Yaskawa INFORM job: u_tourne3TRJ3.JBI

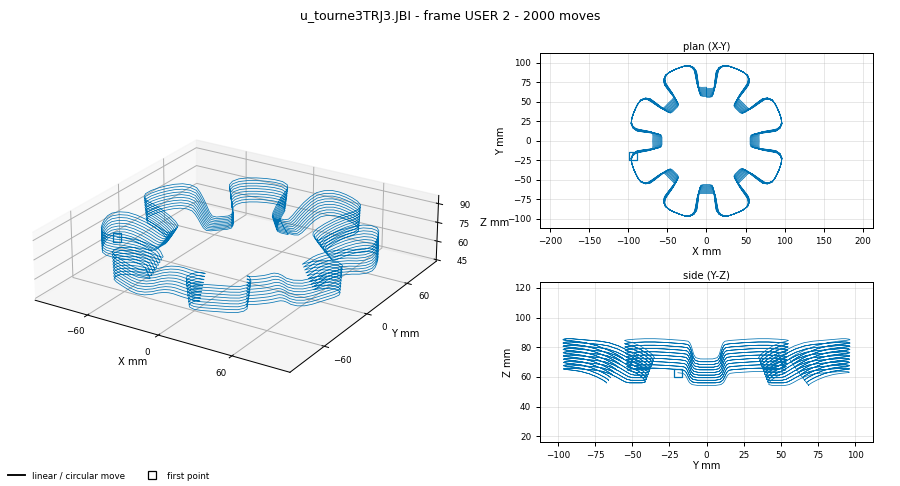
[picture p0: tool path of u_tourne3TRJ3.JBI in frame USER 2, 2000 of 2000 moves have a stored position in this frame; points joined in program order, loops and branches not executed]
/JOB
//NAME u_tourne3TRJ3
///FOLDERNAME DEMO
//POS
///NPOS 2000,0,2000,0,0,0
///USER 2
///TOOL 7
///POSTYPE USER
///RECTAN
///RCONF 1,0,0,0,0,0,0,0,0,0,0,0,0,0,0,0,0,0,0,0,0,0,0,0
C00000=-94.423,-19.246,62.877,176.5198,-3.5287,-10788.4794
C00001=-90.636,-15.942,62.469,172.2266,-2.1131,-10790.0243
C00002=-85.405,-14.621,61.698,172.0565,-0.4508,-10790.2854
C00003=-79.780,-13.569,60.151,173.8939,-0.2961,-10790.3475
C00004=-74.809,-12.586,58.158,176.9112,-0.2537,-10790.4499
C00005=-71.127,-11.507,56.252,-176.4195,0.6994,-10790.8103
C00006=-69.044,-9.699,54.888,-160.3569,24.2302,-10792.0037
C00007=-68.619,-6.200,54.350,-174.8933,38.1355,-10794.8371
C00008=-68.781,-2.945,54.326,179.7056,38.7871,-10797.5483
C00009=-68.843,0.000,54.342,180.0000,38.7770,-10800.0000
C00010=-68.781,2.945,54.326,-179.7056,38.7871,-10802.4517
C00011=-68.619,6.200,54.350,174.8933,38.1355,-10805.1629
C00012=-69.044,9.699,54.888,160.3561,24.2357,-10807.9963
C00013=-71.127,11.507,56.252,176.4195,0.6994,-10809.1897
C00014=-74.809,12.586,58.158,-176.9112,-0.2537,-10809.5501
C00015=-79.780,13.569,60.151,-173.8939,-0.2961,-10809.6525
C00016=-85.405,14.621,61.698,-172.0565,-0.4508,-10809.7146
C00017=-90.636,15.942,62.469,-172.2266,-2.1131,-10809.9757
C00018=-94.423,19.246,62.877,-176.5198,-3.5287,-10811.5206
C00019=-96.154,24.159,63.210,-179.1544,-2.3288,-10814.1038
C00020=-95.429,29.718,63.547,-179.9995,-0.1559,-10817.2974
C00021=-93.512,35.416,63.770,-179.9993,-0.0181,-10820.7433
C00022=-91.166,41.080,63.770,-179.9982,-0.0180,-10824.2566
C00023=-88.493,46.465,63.547,179.9980,-0.1564,-10827.7026
C00024=-85.074,50.908,63.210,179.1554,-2.3286,-10830.8962
C00025=-80.376,53.158,62.877,176.5237,-3.5316,-10833.4793
C00026=-75.362,52.817,62.469,172.2314,-2.1139,-10835.0245
C00027=-70.729,50.052,61.698,172.0558,-0.4490,-10835.2855
C00028=-66.007,46.818,60.151,173.8890,-0.2958,-10835.3476
C00029=-61.798,43.998,58.158,176.9122,-0.2494,-10835.4495
C00030=-58.431,42.158,56.252,-176.4248,0.6998,-10835.8105
C00031=-55.679,41.963,54.888,-160.3550,24.2338,-10837.0038
C00032=-52.905,44.137,54.350,-174.8913,38.1376,-10839.8372
C00033=-50.718,46.553,54.326,179.7087,38.7878,-10842.5482
C00034=-48.679,48.679,54.342,179.9948,38.7763,-10845.0000
C00035=-46.553,50.718,54.326,-179.7087,38.7878,-10847.4518
C00036=-44.137,52.905,54.350,174.8913,38.1376,-10850.1628
C00037=-41.963,55.680,54.888,160.3548,24.2336,-10852.9966
C00038=-42.158,58.431,56.252,176.4248,0.6998,-10854.1895
C00039=-43.998,61.798,58.158,-176.9122,-0.2494,-10854.5505
C00040=-46.818,66.007,60.151,-173.8890,-0.2958,-10854.6524
C00041=-50.052,70.729,61.698,-172.0558,-0.4490,-10854.7145
C00042=-52.817,75.362,62.469,-172.2314,-2.1139,-10854.9755
C00043=-53.158,80.376,62.877,-176.5237,-3.5316,-10856.5207
C00044=-50.908,85.074,63.210,-179.1554,-2.3286,-10859.1038
C00045=-46.465,88.493,63.547,-179.9980,-0.1564,-10862.2974
C00046=-41.080,91.166,63.770,179.9982,-0.0180,-10865.7434
C00047=-35.416,93.512,63.770,179.9993,-0.0181,-10869.2567
C00048=-29.718,95.429,63.547,179.9995,-0.1559,-10872.7026
C00049=-24.159,96.154,63.210,179.1544,-2.3288,-10875.8962
C00050=-19.246,94.423,62.877,176.5198,-3.5287,-10878.4794
C00051=-15.942,90.636,62.469,172.2266,-2.1131,-10880.0243
C00052=-14.621,85.405,61.698,172.0565,-0.4508,-10880.2854
C00053=-13.569,79.780,60.151,173.8939,-0.2961,-10880.3475
C00054=-12.586,74.809,58.158,176.9112,-0.2537,-10880.4499
C00055=-11.507,71.127,56.252,-176.4195,0.6994,-10880.8103
C00056=-9.699,69.044,54.888,-160.3561,24.2357,-10882.0037
C00057=-6.200,68.619,54.350,-174.8933,38.1355,-10884.8371
C00058=-2.945,68.781,54.326,179.7056,38.7871,-10887.5483
C00059=0.000,68.843,54.342,180.0000,38.7770,-10890.0000
C00060=0.000,67.469,56.061,180.0000,38.4594,-10890.0000
C00061=2.820,67.413,56.044,-179.6998,38.4717,-10892.3954
C00062=5.989,67.263,56.069,174.6494,37.7561,-10895.0881
C00063=9.441,67.734,56.637,160.4399,22.8847,-10897.9350
C00064=11.191,69.937,58.076,177.3917,0.4478,-10899.0911
C00065=12.227,73.809,60.085,-176.5319,-0.2393,-10899.4060
C00066=13.183,79.025,62.181,-173.7887,-0.2511,-10899.4709
C00067=14.211,84.918,63.804,-172.0889,-0.3684,-10899.5004
C00068=15.500,90.396,64.610,-172.2474,-1.9783,-10899.7298
C00069=18.832,94.373,65.037,-176.4691,-3.4890,-10901.2851
C00070=23.832,96.213,65.385,-179.1427,-2.3150,-10903.9122
C00071=29.513,95.497,65.736,-179.9981,-0.1613,-10907.1736
C00072=35.347,93.539,65.969,-179.9993,-0.0181,-10910.7008
C00073=41.148,91.136,65.969,-179.9981,-0.0180,-10914.2992
C00074=46.658,88.395,65.736,179.9983,-0.1564,-10917.8267
C00075=51.181,84.885,65.385,179.1465,-2.3148,-10921.0877
C00076=53.416,80.048,65.037,176.4667,-3.4903,-10923.7152
C00077=52.959,74.880,64.610,172.2446,-1.9818,-10925.2699
C00078=49.997,70.095,63.804,172.0881,-0.3719,-10925.4993
C00079=46.557,65.200,62.181,173.7887,-0.2530,-10925.5293
C00080=43.545,60.837,60.085,176.5334,-0.2396,-10925.5938
C00081=41.540,57.367,58.076,-177.3875,0.4483,-10925.9087
C00082=41.220,54.571,56.637,-160.4399,22.8842,-10927.0654
C00083=43.327,51.796,56.069,-174.6518,37.7544,-10929.9123
C00084=45.674,49.662,56.044,179.7031,38.4687,-10932.6047
C00085=47.708,47.708,56.061,-180.0000,38.4581,-10935.0000
C00086=49.662,45.674,56.044,-179.7031,38.4687,-10937.3953
C00087=51.797,43.327,56.069,174.6514,37.7543,-10940.0883
C00088=54.571,41.220,56.637,160.4399,22.8842,-10942.9346
C00089=57.367,41.540,58.076,177.3875,0.4483,-10944.0913
C00090=60.837,43.545,60.085,-176.5334,-0.2396,-10944.4062
C00091=65.200,46.557,62.181,-173.7887,-0.2530,-10944.4707
C00092=70.095,49.997,63.804,-172.0881,-0.3719,-10944.5007
C00093=74.880,52.959,64.610,-172.2446,-1.9818,-10944.7301
C00094=80.048,53.416,65.037,-176.4667,-3.4903,-10946.2848
C00095=84.885,51.181,65.385,-179.1465,-2.3148,-10948.9123
C00096=88.395,46.658,65.736,-179.9983,-0.1564,-10952.1733
C00097=91.136,41.148,65.969,179.9981,-0.0180,-10955.7008
C00098=93.539,35.347,65.969,179.9993,-0.0181,-10959.2992
C00099=95.497,29.513,65.736,179.9981,-0.1613,-10962.8264
C00100=96.213,23.832,65.385,179.1427,-2.3150,-10966.0878
C00101=94.373,18.832,65.037,176.4691,-3.4890,-10968.7149
C00102=90.396,15.500,64.610,172.2474,-1.9783,-10970.2702
C00103=84.918,14.211,63.804,172.0889,-0.3684,-10970.4996
C00104=79.025,13.183,62.181,173.7887,-0.2511,-10970.5291
C00105=73.809,12.227,60.085,176.5319,-0.2393,-10970.5940
C00106=69.937,11.191,58.076,-177.3917,0.4478,-10970.9089
C00107=67.734,9.441,56.637,-160.4399,22.8847,-10972.0650
C00108=67.263,5.989,56.069,-174.6494,37.7561,-10974.9119
C00109=67.413,2.820,56.044,179.6998,38.4717,-10977.6046
C00110=67.469,0.000,56.061,-180.0000,38.4594,-10980.0000
C00111=67.413,-2.820,56.044,-179.6998,38.4717,-10982.3954
C00112=67.263,-5.989,56.069,174.6494,37.7561,-10985.0881
C00113=67.734,-9.441,56.637,160.4399,22.8847,-10987.9350
C00114=69.937,-11.191,58.076,177.3917,0.4478,-10989.0911
C00115=73.809,-12.227,60.085,-176.5319,-0.2393,-10989.4060
C00116=79.025,-13.183,62.181,-173.7887,-0.2511,-10989.4709
C00117=84.918,-14.211,63.804,-172.0889,-0.3684,-10989.5004
C00118=90.396,-15.500,64.610,-172.2474,-1.9783,-10989.7298
C00119=94.373,-18.832,65.037,-176.4691,-3.4890,-10991.2851
C00120=96.213,-23.832,65.385,-179.1427,-2.3150,-10993.9122
C00121=95.497,-29.513,65.736,-179.9981,-0.1613,-10997.1736
C00122=93.539,-35.347,65.969,-179.9993,-0.0181,-11000.7008
C00123=91.136,-41.148,65.969,-179.9981,-0.0180,-11004.2992
C00124=88.395,-46.658,65.736,179.9983,-0.1564,-11007.8267
C00125=84.885,-51.181,65.385,179.1465,-2.3148,-11011.0877
C00126=80.048,-53.416,65.037,176.4667,-3.4903,-11013.7152
C00127=74.880,-52.959,64.610,172.2446,-1.9818,-11015.2699
C00128=70.095,-49.997,63.804,172.0881,-0.3719,-11015.4993
C00129=65.200,-46.557,62.181,173.7887,-0.2530,-11015.5293
C00130=60.837,-43.545,60.085,176.5334,-0.2396,-11015.5938
C00131=57.367,-41.540,58.076,-177.3875,0.4483,-11015.9087
C00132=54.571,-41.220,56.637,-160.4399,22.8842,-11017.0654
C00133=51.796,-43.327,56.069,-174.6518,37.7544,-11019.9123
C00134=49.662,-45.674,56.044,179.7031,38.4687,-11022.6047
C00135=47.708,-47.708,56.061,-180.0000,38.4581,-11025.0000
C00136=45.674,-49.662,56.044,-179.7031,38.4687,-11027.3953
C00137=43.327,-51.797,56.069,174.6514,37.7543,-11030.0883
C00138=41.220,-54.571,56.637,160.4399,22.8842,-11032.9346
C00139=41.540,-57.367,58.076,177.3875,0.4483,-11034.0913
C00140=43.545,-60.837,60.085,-176.5334,-0.2396,-11034.4062
C00141=46.557,-65.200,62.181,-173.7887,-0.2530,-11034.4707
C00142=49.997,-70.095,63.804,-172.0881,-0.3719,-11034.5007
C00143=52.959,-74.880,64.610,-172.2446,-1.9818,-11034.7301
C00144=53.416,-80.048,65.037,-176.4667,-3.4903,-11036.2848
C00145=51.181,-84.885,65.385,-179.1465,-2.3148,-11038.9123
C00146=46.658,-88.395,65.736,-179.9983,-0.1564,-11042.1733
C00147=41.148,-91.136,65.969,179.9981,-0.0180,-11045.7008
C00148=35.347,-93.539,65.969,179.9993,-0.0181,-11049.2992
C00149=29.513,-95.497,65.736,179.9981,-0.1613,-11052.8264
C00150=23.832,-96.213,65.385,179.1427,-2.3150,-11056.0878
C00151=18.832,-94.373,65.037,176.4691,-3.4890,-11058.7149
C00152=15.500,-90.396,64.610,172.2474,-1.9783,-11060.2702
C00153=14.211,-84.918,63.804,172.0889,-0.3684,-11060.4996
C00154=13.183,-79.025,62.181,173.7887,-0.2511,-11060.5291
C00155=12.227,-73.809,60.085,176.5319,-0.2393,-11060.5940
C00156=11.191,-69.937,58.076,-177.3917,0.4478,-11060.9089
C00157=9.441,-67.734,56.637,-160.4399,22.8847,-11062.0650
C00158=5.989,-67.263,56.069,-174.6494,37.7561,-11064.9119
C00159=2.820,-67.413,56.044,179.6998,38.4717,-11067.6046
C00160=0.000,-67.469,56.061,-180.0000,38.4594,-11070.0000
C00161=0.000,-67.469,56.061,-180.0000,38.4594,-11070.0000
C00162=-2.820,-67.413,56.044,-179.6998,38.4717,-11072.3954
C00163=-5.989,-67.263,56.069,174.6494,37.7561,-11075.0881
C00164=-9.441,-67.734,56.637,160.4399,22.8847,-11077.9350
C00165=-11.191,-69.937,58.076,177.3917,0.4478,-11079.0911
C00166=-12.227,-73.809,60.085,-176.5319,-0.2393,-11079.4060
C00167=-13.183,-79.025,62.181,-173.7887,-0.2511,-11079.4709
C00168=-14.211,-84.918,63.804,-172.0889,-0.3684,-11079.5004
C00169=-15.500,-90.396,64.610,-172.2474,-1.9783,-11079.7298
C00170=-18.832,-94.373,65.037,-176.4691,-3.4890,-11081.2851
C00171=-23.832,-96.213,65.385,-179.1427,-2.3150,-11083.9122
C00172=-29.513,-95.497,65.736,-179.9981,-0.1613,-11087.1736
C00173=-35.347,-93.539,65.969,-179.9993,-0.0181,-11090.7008
C00174=-41.148,-91.136,65.969,-179.9981,-0.0180,-11094.2992
C00175=-46.658,-88.395,65.736,179.9983,-0.1564,-11097.8267
C00176=-51.181,-84.885,65.385,179.1465,-2.3148,-11101.0877
C00177=-53.416,-80.048,65.037,176.4667,-3.4903,-11103.7152
C00178=-52.959,-74.880,64.610,172.2446,-1.9818,-11105.2699
C00179=-49.997,-70.095,63.804,172.0881,-0.3719,-11105.4993
C00180=-46.557,-65.200,62.181,173.7887,-0.2530,-11105.5293
C00181=-43.545,-60.837,60.085,176.5334,-0.2396,-11105.5938
C00182=-41.540,-57.367,58.076,-177.3875,0.4483,-11105.9087
C00183=-41.220,-54.571,56.637,-160.4399,22.8842,-11107.0654
C00184=-43.327,-51.796,56.069,-174.6518,37.7544,-11109.9123
C00185=-45.674,-49.662,56.044,179.7031,38.4687,-11112.6047
C00186=-47.708,-47.708,56.061,-180.0000,38.4581,-11115.0000
C00187=-49.662,-45.674,56.044,-179.7031,38.4687,-11117.3953
C00188=-51.797,-43.327,56.069,174.6514,37.7543,-11120.0883
C00189=-54.571,-41.220,56.637,160.4399,22.8842,-11122.9346
C00190=-57.367,-41.540,58.076,177.3875,0.4483,-11124.0913
C00191=-60.837,-43.545,60.085,-176.5334,-0.2396,-11124.4062
C00192=-65.200,-46.557,62.181,-173.7887,-0.2530,-11124.4707
C00193=-70.095,-49.997,63.804,-172.0881,-0.3719,-11124.5007
C00194=-74.880,-52.959,64.610,-172.2446,-1.9818,-11124.7301
C00195=-80.048,-53.416,65.037,-176.4667,-3.4903,-11126.2848
C00196=-84.885,-51.181,65.385,-179.1465,-2.3148,-11128.9123
C00197=-88.395,-46.658,65.736,-179.9983,-0.1564,-11132.1733
C00198=-91.136,-41.148,65.969,179.9981,-0.0180,-11135.7008
C00199=-93.539,-35.347,65.969,179.9993,-0.0181,-11139.2992
C00200=-95.497,-29.513,65.736,179.9981,-0.1613,-11142.8264
C00201=-96.213,-23.832,65.385,179.1427,-2.3150,-11146.0878
C00202=-94.373,-18.832,65.037,176.4691,-3.4890,-11148.7149
C00203=-90.396,-15.500,64.610,172.2474,-1.9783,-11150.2702
C00204=-84.918,-14.211,63.804,172.0889,-0.3684,-11150.4996
C00205=-79.025,-13.183,62.181,173.7887,-0.2511,-11150.5291
C00206=-73.809,-12.227,60.085,176.5319,-0.2393,-11150.5940
C00207=-69.937,-11.191,58.076,-177.3917,0.4478,-11150.9089
C00208=-67.734,-9.441,56.637,-160.4399,22.8847,-11152.0650
C00209=-67.263,-5.989,56.069,-174.6494,37.7561,-11154.9119
C00210=-67.413,-2.820,56.044,179.6998,38.4717,-11157.6046
C00211=-67.469,0.000,56.061,-180.0000,38.4594,-11160.0000
C00212=-67.413,2.820,56.044,-179.6998,38.4717,-11162.3954
C00213=-67.263,5.989,56.069,174.6494,37.7561,-11165.0881
C00214=-67.734,9.441,56.637,160.4399,22.8847,-11167.9350
C00215=-69.937,11.191,58.076,177.3917,0.4478,-11169.0911
C00216=-73.809,12.227,60.085,-176.5319,-0.2393,-11169.4060
C00217=-79.025,13.183,62.181,-173.7887,-0.2511,-11169.4709
C00218=-84.918,14.211,63.804,-172.0889,-0.3684,-11169.5004
C00219=-90.396,15.500,64.610,-172.2474,-1.9783,-11169.7298
C00220=-94.373,18.832,65.037,-176.4691,-3.4890,-11171.2851
C00221=-96.213,23.832,65.385,-179.1427,-2.3150,-11173.9122
C00222=-95.497,29.513,65.736,-179.9981,-0.1613,-11177.1736
C00223=-93.539,35.347,65.969,-179.9993,-0.0181,-11180.7008
C00224=-91.136,41.148,65.969,-179.9981,-0.0180,-11184.2992
C00225=-88.395,46.658,65.736,179.9983,-0.1564,-11187.8267
C00226=-84.885,51.181,65.385,179.1465,-2.3148,-11191.0877
C00227=-80.048,53.416,65.037,176.4667,-3.4903,-11193.7152
C00228=-74.880,52.959,64.610,172.2446,-1.9818,-11195.2699
C00229=-70.095,49.997,63.804,172.0881,-0.3719,-11195.4993
C00230=-65.200,46.557,62.181,173.7887,-0.2530,-11195.5293
C00231=-60.837,43.545,60.085,176.5334,-0.2396,-11195.5938
C00232=-57.367,41.540,58.076,-177.3875,0.4483,-11195.9087
C00233=-54.571,41.220,56.637,-160.4399,22.8842,-11197.0654
C00234=-51.796,43.327,56.069,-174.6518,37.7544,-11199.9123
C00235=-49.662,45.674,56.044,179.7031,38.4687,-11202.6047
C00236=-47.708,47.708,56.061,-180.0000,38.4581,-11205.0000
C00237=-45.674,49.662,56.044,-179.7031,38.4687,-11207.3953
C00238=-43.327,51.797,56.069,174.6514,37.7543,-11210.0883
C00239=-41.220,54.571,56.637,160.4399,22.8842,-11212.9346
C00240=-41.540,57.367,58.076,177.3875,0.4483,-11214.0913
C00241=-43.545,60.837,60.085,-176.5334,-0.2396,-11214.4062
C00242=-46.557,65.200,62.181,-173.7887,-0.2530,-11214.4707
C00243=-49.997,70.095,63.804,-172.0881,-0.3719,-11214.5007
C00244=-52.959,74.880,64.610,-172.2446,-1.9818,-11214.7301
C00245=-53.416,80.048,65.037,-176.4667,-3.4903,-11216.2848
C00246=-51.181,84.885,65.385,-179.1465,-2.3148,-11218.9123
C00247=-46.658,88.395,65.736,-179.9983,-0.1564,-11222.1733
C00248=-41.148,91.136,65.969,179.9981,-0.0180,-11225.7008
C00249=-35.347,93.539,65.969,179.9993,-0.0181,-11229.2992
C00250=-29.513,95.497,65.736,179.9981,-0.1613,-11232.8264
C00251=-23.832,96.213,65.385,179.1427,-2.3150,-11236.0878
C00252=-18.832,94.373,65.037,176.4691,-3.4890,-11238.7149
C00253=-15.500,90.396,64.610,172.2474,-1.9783,-11240.2702
C00254=-14.211,84.918,63.804,172.0889,-0.3684,-11240.4996
C00255=-13.183,79.025,62.181,173.7887,-0.2511,-11240.5291
C00256=-12.227,73.809,60.085,176.5319,-0.2393,-11240.5940
C00257=-11.191,69.937,58.076,-177.3917,0.4478,-11240.9089
C00258=-9.441,67.734,56.637,-160.4399,22.8847,-11242.0650
C00259=-5.989,67.263,56.069,-174.6494,37.7561,-11244.9119
C00260=-2.820,67.413,56.044,179.6998,38.4717,-11247.6046
C00261=0.000,67.469,56.061,180.0000,38.4594,-11250.0000
C00262=0.000,66.107,57.788,180.0000,38.0594,-11250.0000
C00263=2.695,66.055,57.771,-179.6967,38.0667,-11252.3363
C00264=5.779,65.917,57.797,174.4231,37.2903,-11255.0104
C00265=9.185,66.436,58.394,160.6412,21.4973,-11257.8714
C00266=10.880,68.762,59.909,178.2705,0.2602,-11258.9912
C00267=11.874,72.826,62.021,-176.2283,-0.2219,-11259.2604
C00268=12.805,78.288,64.219,-173.7529,-0.2122,-11259.2892
C00269=13.814,84.445,65.915,-172.1933,-0.3031,-11259.2905
C00270=15.073,90.163,66.756,-172.3373,-1.8422,-11259.4907
C00271=18.432,94.325,67.200,-176.4590,-3.4166,-11261.0568
C00272=23.517,96.271,67.561,-179.1417,-2.2803,-11263.7273
C00273=29.315,95.562,67.927,179.9999,-0.1559,-11267.0541
C00274=35.280,93.564,68.167,-179.9993,-0.0181,-11270.6599
C00275=41.213,91.107,68.167,-179.9981,-0.0180,-11274.3400
C00276=46.844,88.301,67.927,179.9986,-0.1564,-11277.9461
C00277=51.445,84.703,67.561,179.1429,-2.2773,-11281.2727
C00278=53.664,79.731,67.200,176.4564,-3.4170,-11283.9430
C00279=53.097,74.413,66.756,172.3397,-1.8459,-11285.5096
C00280=49.944,69.479,65.915,172.1917,-0.3060,-11285.7099
C00281=46.303,64.413,64.219,173.7509,-0.2085,-11285.7103
C00282=43.100,59.892,62.021,176.2254,-0.2229,-11285.7399
C00283=40.929,56.315,59.909,-178.2687,0.2595,-11286.0092
C00284=40.483,53.472,58.394,-160.6426,21.4997,-11287.1289
C00285=42.524,50.697,57.797,-174.4236,37.2887,-11289.9895
C00286=44.802,48.614,57.771,179.6988,38.0662,-11292.6632
C00287=46.745,46.745,57.788,180.0000,38.0574,-11295.0000
C00288=48.613,44.802,57.771,-179.6984,38.0662,-11297.3362
C00289=50.697,42.524,57.797,174.4190,37.2852,-11300.0105
C00290=53.472,40.483,58.395,160.6426,21.4997,-11302.8711
C00291=56.315,40.929,59.909,178.2687,0.2595,-11303.9908
C00292=59.892,43.100,62.021,-176.2254,-0.2229,-11304.2601
C00293=64.413,46.303,64.219,-173.7509,-0.2085,-11304.2897
C00294=69.479,49.944,65.915,-172.1917,-0.3060,-11304.2901
C00295=74.413,53.097,66.756,-172.3397,-1.8459,-11304.4904
C00296=79.731,53.664,67.200,-176.4564,-3.4170,-11306.0570
C00297=84.703,51.445,67.561,-179.1429,-2.2773,-11308.7273
C00298=88.301,46.844,67.927,-179.9986,-0.1564,-11312.0539
C00299=91.107,41.213,68.167,179.9981,-0.0180,-11315.6600
C00300=93.564,35.280,68.167,179.9993,-0.0181,-11319.3401
C00301=95.562,29.315,67.927,-179.9999,-0.1559,-11322.9459
C00302=96.271,23.517,67.561,179.1417,-2.2803,-11326.2727
C00303=94.325,18.432,67.200,176.4590,-3.4166,-11328.9432
C00304=90.163,15.073,66.756,172.3373,-1.8422,-11330.5093
C00305=84.445,13.814,65.915,172.1933,-0.3031,-11330.7095
C00306=78.288,12.805,64.219,173.7529,-0.2122,-11330.7108
C00307=72.826,11.874,62.021,176.2283,-0.2219,-11330.7396
C00308=68.762,10.880,59.909,-178.2705,0.2602,-11331.0088
C00309=66.436,9.185,58.394,-160.6412,21.4973,-11332.1286
C00310=65.917,5.779,57.797,-174.4231,37.2903,-11334.9896
C00311=66.055,2.695,57.771,179.6967,38.0667,-11337.6637
C00312=66.107,0.000,57.788,180.0000,38.0594,-11340.0000
C00313=66.055,-2.695,57.771,-179.6967,38.0667,-11342.3363
C00314=65.917,-5.780,57.797,174.4154,37.2898,-11345.0112
C00315=66.436,-9.185,58.395,160.6412,21.4973,-11347.8714
C00316=68.762,-10.880,59.909,178.2705,0.2602,-11348.9912
C00317=72.826,-11.874,62.021,-176.2283,-0.2219,-11349.2604
C00318=78.288,-12.805,64.219,-173.7529,-0.2122,-11349.2892
C00319=84.445,-13.814,65.915,-172.1933,-0.3031,-11349.2905
C00320=90.163,-15.073,66.756,-172.3373,-1.8422,-11349.4907
C00321=94.325,-18.432,67.200,-176.4590,-3.4166,-11351.0568
C00322=96.271,-23.517,67.561,-179.1417,-2.2803,-11353.7273
C00323=95.562,-29.315,67.927,179.9999,-0.1559,-11357.0541
C00324=93.564,-35.280,68.167,-179.9993,-0.0181,-11360.6599
C00325=91.107,-41.213,68.167,-179.9981,-0.0180,-11364.3400
C00326=88.301,-46.844,67.927,179.9986,-0.1564,-11367.9461
C00327=84.703,-51.445,67.561,179.1429,-2.2773,-11371.2727
C00328=79.731,-53.664,67.200,176.4564,-3.4170,-11373.9430
C00329=74.413,-53.097,66.756,172.3397,-1.8459,-11375.5096
C00330=69.479,-49.944,65.915,172.1917,-0.3060,-11375.7099
C00331=64.413,-46.303,64.219,173.7509,-0.2085,-11375.7103
C00332=59.892,-43.100,62.021,176.2254,-0.2229,-11375.7399
C00333=56.315,-40.929,59.909,-178.2687,0.2595,-11376.0092
C00334=53.472,-40.483,58.394,-160.6426,21.4997,-11377.1289
C00335=50.697,-42.524,57.797,-174.4236,37.2887,-11379.9895
C00336=48.614,-44.802,57.771,179.6988,38.0662,-11382.6632
C00337=46.745,-46.745,57.788,180.0000,38.0574,-11385.0000
C00338=44.802,-48.613,57.771,-179.6984,38.0662,-11387.3362
C00339=42.524,-50.697,57.797,174.4190,37.2852,-11390.0105
C00340=40.483,-53.472,58.395,160.6426,21.4997,-11392.8711
C00341=40.929,-56.315,59.909,178.2687,0.2595,-11393.9908
C00342=43.100,-59.892,62.021,-176.2254,-0.2229,-11394.2601
C00343=46.303,-64.413,64.219,-173.7509,-0.2085,-11394.2897
C00344=49.944,-69.479,65.915,-172.1917,-0.3060,-11394.2901
C00345=53.097,-74.413,66.756,-172.3397,-1.8459,-11394.4904
C00346=53.664,-79.731,67.200,-176.4564,-3.4170,-11396.0570
C00347=51.445,-84.703,67.561,-179.1429,-2.2773,-11398.7273
C00348=46.844,-88.301,67.927,-179.9986,-0.1564,-11402.0539
C00349=41.213,-91.107,68.167,179.9981,-0.0180,-11405.6600
C00350=35.280,-93.564,68.167,179.9993,-0.0181,-11409.3401
C00351=29.315,-95.562,67.927,-179.9999,-0.1559,-11412.9459
C00352=23.517,-96.271,67.561,179.1417,-2.2803,-11416.2727
C00353=18.432,-94.325,67.200,176.4590,-3.4166,-11418.9432
C00354=15.073,-90.163,66.756,172.3373,-1.8422,-11420.5093
C00355=13.814,-84.445,65.915,172.1933,-0.3031,-11420.7095
C00356=12.805,-78.288,64.219,173.7529,-0.2122,-11420.7108
C00357=11.874,-72.826,62.021,176.2283,-0.2219,-11420.7396
C00358=10.880,-68.762,59.909,-178.2705,0.2602,-11421.0088
C00359=9.185,-66.436,58.394,-160.6412,21.4973,-11422.1286
C00360=5.779,-65.917,57.797,-174.4231,37.2903,-11424.9896
C00361=2.695,-66.055,57.771,179.6967,38.0667,-11427.6637
C00362=0.000,-66.107,57.788,-180.0000,38.0594,-11430.0000
C00363=0.000,-66.107,57.788,-180.0000,38.0594,-11430.0000
C00364=-2.695,-66.055,57.771,-179.6967,38.0667,-11432.3363
C00365=-5.780,-65.917,57.797,174.4154,37.2898,-11435.0112
C00366=-9.185,-66.436,58.395,160.6412,21.4973,-11437.8714
C00367=-10.880,-68.762,59.909,178.2705,0.2602,-11438.9912
C00368=-11.874,-72.826,62.021,-176.2283,-0.2219,-11439.2604
C00369=-12.805,-78.288,64.219,-173.7529,-0.2122,-11439.2892
C00370=-13.814,-84.445,65.915,-172.1933,-0.3031,-11439.2905
C00371=-15.073,-90.163,66.756,-172.3373,-1.8422,-11439.4907
C00372=-18.432,-94.325,67.200,-176.4590,-3.4166,-11441.0568
C00373=-23.517,-96.271,67.561,-179.1417,-2.2803,-11443.7273
C00374=-29.315,-95.562,67.927,179.9999,-0.1559,-11447.0541
C00375=-35.280,-93.564,68.167,-179.9993,-0.0181,-11450.6599
C00376=-41.213,-91.107,68.167,-179.9981,-0.0180,-11454.3400
C00377=-46.844,-88.301,67.927,179.9986,-0.1564,-11457.9461
C00378=-51.445,-84.703,67.561,179.1429,-2.2773,-11461.2727
C00379=-53.664,-79.731,67.200,176.4564,-3.4170,-11463.9430
C00380=-53.097,-74.413,66.756,172.3397,-1.8459,-11465.5096
C00381=-49.944,-69.479,65.915,172.1917,-0.3060,-11465.7099
C00382=-46.303,-64.413,64.219,173.7509,-0.2085,-11465.7103
C00383=-43.100,-59.892,62.021,176.2254,-0.2229,-11465.7399
C00384=-40.929,-56.315,59.909,-178.2687,0.2595,-11466.0092
C00385=-40.483,-53.472,58.394,-160.6426,21.4997,-11467.1289
C00386=-42.524,-50.697,57.797,-174.4236,37.2887,-11469.9895
C00387=-44.802,-48.614,57.771,179.6988,38.0662,-11472.6632
C00388=-46.745,-46.745,57.788,-180.0000,38.0574,-11475.0000
C00389=-48.613,-44.802,57.771,-179.6984,38.0662,-11477.3362
C00390=-50.697,-42.524,57.797,174.4190,37.2852,-11480.0105
C00391=-53.472,-40.483,58.395,160.6426,21.4997,-11482.8711
C00392=-56.315,-40.929,59.909,178.2687,0.2595,-11483.9908
C00393=-59.892,-43.100,62.021,-176.2254,-0.2229,-11484.2601
C00394=-64.413,-46.303,64.219,-173.7509,-0.2085,-11484.2897
C00395=-69.479,-49.944,65.915,-172.1917,-0.3060,-11484.2901
C00396=-74.413,-53.097,66.756,-172.3397,-1.8459,-11484.4904
C00397=-79.731,-53.664,67.200,-176.4564,-3.4170,-11486.0570
C00398=-84.703,-51.445,67.561,-179.1429,-2.2773,-11488.7273
C00399=-88.301,-46.844,67.927,-179.9986,-0.1564,-11492.0539
C00400=-91.107,-41.213,68.167,179.9981,-0.0180,-11495.6600
C00401=-93.564,-35.280,68.167,179.9993,-0.0181,-11499.3401
C00402=-95.562,-29.315,67.927,-179.9999,-0.1559,-11502.9459
C00403=-96.271,-23.517,67.561,179.1417,-2.2803,-11506.2727
C00404=-94.325,-18.432,67.200,176.4590,-3.4166,-11508.9432
C00405=-90.163,-15.073,66.756,172.3373,-1.8422,-11510.5093
C00406=-84.445,-13.814,65.915,172.1933,-0.3031,-11510.7095
C00407=-78.288,-12.805,64.219,173.7529,-0.2122,-11510.7108
C00408=-72.826,-11.874,62.021,176.2283,-0.2219,-11510.7396
C00409=-68.762,-10.880,59.909,-178.2705,0.2602,-11511.0088
C00410=-66.436,-9.185,58.394,-160.6412,21.4973,-11512.1286
C00411=-65.917,-5.779,57.797,-174.4231,37.2903,-11514.9896
C00412=-66.055,-2.695,57.771,179.6967,38.0667,-11517.6637
C00413=-66.107,0.000,57.788,-180.0000,38.0594,-11520.0000
C00414=-66.055,2.695,57.771,-179.6967,38.0667,-11522.3363
C00415=-65.917,5.780,57.797,174.4154,37.2898,-11525.0112
C00416=-66.436,9.185,58.395,160.6412,21.4973,-11527.8714
C00417=-68.762,10.880,59.909,178.2705,0.2602,-11528.9912
C00418=-72.826,11.874,62.021,-176.2283,-0.2219,-11529.2604
C00419=-78.288,12.805,64.219,-173.7529,-0.2122,-11529.2892
C00420=-84.445,13.814,65.915,-172.1933,-0.3031,-11529.2905
C00421=-90.163,15.073,66.756,-172.3373,-1.8422,-11529.4907
C00422=-94.325,18.432,67.200,-176.4590,-3.4166,-11531.0568
C00423=-96.271,23.517,67.561,-179.1417,-2.2803,-11533.7273
C00424=-95.562,29.315,67.927,179.9999,-0.1559,-11537.0541
C00425=-93.564,35.280,68.167,-179.9993,-0.0181,-11540.6599
C00426=-91.107,41.213,68.167,-179.9981,-0.0180,-11544.3400
C00427=-88.301,46.844,67.927,179.9986,-0.1564,-11547.9461
C00428=-84.703,51.445,67.561,179.1429,-2.2773,-11551.2727
C00429=-79.731,53.664,67.200,176.4564,-3.4170,-11553.9430
C00430=-74.413,53.097,66.756,172.3397,-1.8459,-11555.5096
C00431=-69.479,49.944,65.915,172.1917,-0.3060,-11555.7099
C00432=-64.413,46.303,64.219,173.7509,-0.2085,-11555.7103
C00433=-59.892,43.100,62.021,176.2254,-0.2229,-11555.7399
C00434=-56.315,40.929,59.909,-178.2687,0.2595,-11556.0092
C00435=-53.472,40.483,58.394,-160.6426,21.4997,-11557.1289
C00436=-50.697,42.524,57.797,-174.4236,37.2887,-11559.9895
C00437=-48.614,44.802,57.771,179.6988,38.0662,-11562.6632
C00438=-46.745,46.745,57.788,-180.0000,38.0574,-11565.0000
C00439=-44.802,48.613,57.771,-179.6984,38.0662,-11567.3362
C00440=-42.524,50.697,57.797,174.4190,37.2852,-11570.0105
C00441=-40.483,53.472,58.395,160.6426,21.4997,-11572.8711
C00442=-40.929,56.315,59.909,178.2687,0.2595,-11573.9908
C00443=-43.100,59.892,62.021,-176.2254,-0.2229,-11574.2601
C00444=-46.303,64.413,64.219,-173.7509,-0.2085,-11574.2897
C00445=-49.944,69.479,65.915,-172.1917,-0.3060,-11574.2901
C00446=-53.097,74.413,66.756,-172.3397,-1.8459,-11574.4904
C00447=-53.664,79.731,67.200,-176.4564,-3.4170,-11576.0570
C00448=-51.445,84.703,67.561,-179.1429,-2.2773,-11578.7273
C00449=-46.844,88.301,67.927,-179.9986,-0.1564,-11582.0539
C00450=-41.213,91.107,68.167,179.9981,-0.0180,-11585.6600
C00451=-35.280,93.564,68.167,179.9993,-0.0181,-11589.3401
C00452=-29.315,95.562,67.927,-179.9999,-0.1559,-11592.9459
C00453=-23.517,96.271,67.561,179.1417,-2.2803,-11596.2727
C00454=-18.432,94.325,67.200,176.4590,-3.4166,-11598.9432
C00455=-15.073,90.163,66.756,172.3373,-1.8422,-11600.5093
C00456=-13.814,84.445,65.915,172.1933,-0.3031,-11600.7095
C00457=-12.805,78.288,64.219,173.7529,-0.2122,-11600.7108
C00458=-11.874,72.826,62.021,176.2283,-0.2219,-11600.7396
C00459=-10.880,68.762,59.909,-178.2705,0.2602,-11601.0088
C00460=-9.185,66.436,58.395,-160.6412,21.4973,-11602.1286
C00461=-5.780,65.917,57.797,-174.4154,37.2898,-11604.9888
C00462=-2.695,66.055,57.771,179.6967,38.0667,-11607.6637
C00463=0.000,66.107,57.788,-180.0000,38.0594,-11610.0000
C00464=0.000,64.758,59.526,-180.0000,37.5735,-11610.0000
C00465=2.572,64.710,59.508,-179.6979,37.5837,-11612.2761
C00466=5.572,64.584,59.535,174.2146,36.7296,-11614.9310
C00467=8.932,65.152,60.163,160.9703,20.0908,-11617.8063
C00468=10.572,67.603,61.754,179.0583,0.1253,-11618.8881
C00469=11.527,71.864,63.969,-175.9897,-0.1992,-11619.1126
C00470=12.439,77.571,66.266,-173.7747,-0.1711,-11619.1102
C00471=13.430,83.988,68.033,-172.3612,-0.2407,-11619.0849
C00472=14.662,89.940,68.906,-172.5060,-1.7115,-11619.2589
C00473=18.048,94.279,69.366,-176.4898,-3.3102,-11620.8371
C00474=23.215,96.325,69.740,-179.1510,-2.2246,-11623.5503
C00475=29.126,95.625,70.117,179.9996,-0.1559,-11626.9400
C00476=35.216,93.589,70.366,-179.9993,-0.0181,-11630.6205
C00477=41.276,91.079,70.366,-179.9981,-0.0180,-11634.3795
C00478=47.022,88.212,70.117,179.9990,-0.1564,-11638.0601
C00479=51.697,84.528,69.740,179.1554,-2.2229,-11641.4498
C00480=53.903,79.427,69.366,176.4883,-3.3136,-11644.1627
C00481=53.229,73.964,68.906,172.5034,-1.7072,-11645.7411
C00482=49.892,68.885,68.033,172.3610,-0.2408,-11645.9150
C00483=46.056,63.647,66.266,173.7731,-0.1698,-11645.8901
C00484=42.664,58.966,63.969,175.9921,-0.2034,-11645.8871
C00485=40.327,55.279,61.754,-179.0540,0.1227,-11646.1114
C00486=39.754,52.385,60.163,-160.9694,20.0893,-11647.1942
C00487=41.728,49.608,59.535,-174.2183,36.7311,-11650.0690
C00488=43.938,47.576,59.508,179.6961,37.5811,-11652.7235
C00489=45.791,45.791,59.526,-180.0000,37.5739,-11655.0000
C00490=47.575,43.938,59.508,-179.6957,37.5811,-11657.2759
C00491=49.608,41.728,59.535,174.2083,36.7306,-11659.9310
C00492=52.385,39.754,60.163,160.9694,20.0893,-11662.8058
C00493=55.279,40.327,61.754,179.0540,0.1227,-11663.8886
C00494=58.966,42.664,63.969,-175.9921,-0.2034,-11664.1129
C00495=63.647,46.056,66.266,-173.7731,-0.1698,-11664.1099
C00496=68.885,49.892,68.033,-172.3610,-0.2408,-11664.0850
C00497=73.964,53.229,68.906,-172.5034,-1.7072,-11664.2589
C00498=79.427,53.903,69.366,-176.4883,-3.3136,-11665.8373
C00499=84.528,51.697,69.740,-179.1554,-2.2229,-11668.5502
C00500=88.212,47.022,70.117,-179.9990,-0.1564,-11671.9399
C00501=91.079,41.276,70.366,179.9981,-0.0180,-11675.6205
C00502=93.589,35.216,70.366,179.9993,-0.0181,-11679.3795
C00503=95.625,29.126,70.117,-179.9996,-0.1559,-11683.0600
C00504=96.325,23.215,69.740,179.1510,-2.2246,-11686.4497
C00505=94.279,18.048,69.366,176.4898,-3.3102,-11689.1629
C00506=89.940,14.662,68.906,172.5060,-1.7115,-11690.7411
C00507=83.988,13.430,68.033,172.3612,-0.2407,-11690.9151
C00508=77.571,12.439,66.266,173.7747,-0.1711,-11690.8898
C00509=71.864,11.527,63.969,175.9897,-0.1992,-11690.8874
C00510=67.603,10.572,61.754,-179.0583,0.1253,-11691.1119
C00511=65.152,8.932,60.163,-160.9703,20.0908,-11692.1937
C00512=64.584,5.572,59.535,-174.2146,36.7296,-11695.0690
C00513=64.710,2.572,59.508,179.6979,37.5837,-11697.7239
C00514=64.758,0.000,59.526,180.0000,37.5735,-11700.0000
C00515=64.710,-2.572,59.508,-179.6979,37.5837,-11702.2761
C00516=64.584,-5.572,59.535,174.2146,36.7296,-11704.9310
C00517=65.152,-8.932,60.163,160.9703,20.0908,-11707.8063
C00518=67.603,-10.572,61.754,179.0583,0.1253,-11708.8881
C00519=71.864,-11.527,63.969,-175.9897,-0.1992,-11709.1126
C00520=77.571,-12.439,66.266,-173.7747,-0.1711,-11709.1102
C00521=83.988,-13.430,68.033,-172.3612,-0.2407,-11709.0849
C00522=89.940,-14.662,68.906,-172.5060,-1.7115,-11709.2589
C00523=94.279,-18.048,69.366,-176.4898,-3.3102,-11710.8371
C00524=96.325,-23.215,69.740,-179.1510,-2.2246,-11713.5503
C00525=95.625,-29.126,70.117,179.9996,-0.1559,-11716.9400
C00526=93.589,-35.216,70.366,-179.9993,-0.0181,-11720.6205
C00527=91.079,-41.276,70.366,-179.9981,-0.0180,-11724.3795
C00528=88.212,-47.022,70.117,179.9990,-0.1564,-11728.0601
C00529=84.528,-51.697,69.740,179.1554,-2.2229,-11731.4498
C00530=79.427,-53.903,69.366,176.4883,-3.3136,-11734.1627
C00531=73.964,-53.229,68.906,172.5034,-1.7072,-11735.7411
C00532=68.885,-49.892,68.033,172.3610,-0.2408,-11735.9150
C00533=63.647,-46.056,66.266,173.7731,-0.1698,-11735.8901
C00534=58.966,-42.664,63.969,175.9921,-0.2034,-11735.8871
C00535=55.279,-40.327,61.754,-179.0540,0.1227,-11736.1114
C00536=52.385,-39.754,60.163,-160.9694,20.0893,-11737.1942
C00537=49.608,-41.728,59.535,-174.2183,36.7311,-11740.0690
C00538=47.576,-43.938,59.508,179.6961,37.5811,-11742.7235
C00539=45.791,-45.791,59.526,180.0000,37.5739,-11745.0000
C00540=43.938,-47.575,59.508,-179.6957,37.5811,-11747.2759
C00541=41.728,-49.608,59.535,174.2083,36.7306,-11749.9310
C00542=39.754,-52.385,60.163,160.9694,20.0893,-11752.8058
C00543=40.327,-55.279,61.754,179.0540,0.1227,-11753.8886
C00544=42.664,-58.966,63.969,-175.9921,-0.2034,-11754.1129
C00545=46.056,-63.647,66.266,-173.7731,-0.1698,-11754.1099
C00546=49.892,-68.885,68.033,-172.3610,-0.2408,-11754.0850
C00547=53.229,-73.964,68.906,-172.5034,-1.7072,-11754.2589
C00548=53.903,-79.427,69.366,-176.4883,-3.3136,-11755.8373
C00549=51.697,-84.528,69.740,-179.1554,-2.2229,-11758.5502
C00550=47.022,-88.212,70.117,-179.9990,-0.1564,-11761.9399
C00551=41.276,-91.079,70.366,179.9981,-0.0180,-11765.6205
C00552=35.216,-93.589,70.366,179.9993,-0.0181,-11769.3795
C00553=29.126,-95.625,70.117,-179.9996,-0.1559,-11773.0600
C00554=23.215,-96.325,69.740,179.1510,-2.2246,-11776.4497
C00555=18.048,-94.279,69.366,176.4898,-3.3102,-11779.1629
C00556=14.662,-89.940,68.906,172.5060,-1.7115,-11780.7411
C00557=13.430,-83.988,68.033,172.3612,-0.2407,-11780.9151
C00558=12.439,-77.571,66.266,173.7747,-0.1711,-11780.8898
C00559=11.527,-71.864,63.969,175.9897,-0.1992,-11780.8874
C00560=10.572,-67.603,61.754,-179.0583,0.1253,-11781.1119
C00561=8.932,-65.152,60.163,-160.9703,20.0908,-11782.1937
C00562=5.572,-64.584,59.535,-174.2146,36.7296,-11785.0690
C00563=2.572,-64.710,59.508,179.6979,37.5837,-11787.7239
C00564=0.000,-64.758,59.526,180.0000,37.5735,-11790.0000
C00565=0.000,-64.758,59.526,180.0000,37.5735,-11790.0000
C00566=-2.572,-64.710,59.508,-179.6979,37.5837,-11792.2761
C00567=-5.572,-64.584,59.535,174.2146,36.7296,-11794.9310
C00568=-8.932,-65.152,60.163,160.9703,20.0908,-11797.8063
C00569=-10.572,-67.603,61.754,179.0583,0.1253,-11798.8881
C00570=-11.527,-71.864,63.969,-175.9897,-0.1992,-11799.1126
C00571=-12.439,-77.571,66.266,-173.7747,-0.1711,-11799.1102
C00572=-13.430,-83.988,68.033,-172.3612,-0.2407,-11799.0849
C00573=-14.662,-89.940,68.906,-172.5060,-1.7115,-11799.2589
C00574=-18.048,-94.279,69.366,-176.4898,-3.3102,-11800.8371
C00575=-23.215,-96.325,69.740,-179.1510,-2.2246,-11803.5503
C00576=-29.126,-95.625,70.117,179.9996,-0.1559,-11806.9400
C00577=-35.216,-93.589,70.366,-179.9993,-0.0181,-11810.6205
C00578=-41.276,-91.079,70.366,-179.9981,-0.0180,-11814.3795
C00579=-47.022,-88.212,70.117,179.9990,-0.1564,-11818.0601
C00580=-51.697,-84.528,69.740,179.1554,-2.2229,-11821.4498
C00581=-53.903,-79.427,69.366,176.4883,-3.3136,-11824.1627
C00582=-53.229,-73.964,68.906,172.5034,-1.7072,-11825.7411
C00583=-49.892,-68.885,68.033,172.3610,-0.2408,-11825.9150
C00584=-46.056,-63.647,66.266,173.7731,-0.1698,-11825.8901
C00585=-42.664,-58.966,63.969,175.9921,-0.2034,-11825.8871
C00586=-40.327,-55.279,61.754,-179.0540,0.1227,-11826.1114
C00587=-39.754,-52.385,60.163,-160.9694,20.0893,-11827.1942
C00588=-41.728,-49.608,59.535,-174.2183,36.7311,-11830.0690
C00589=-43.938,-47.576,59.508,179.6961,37.5811,-11832.7235
C00590=-45.791,-45.791,59.526,180.0000,37.5739,-11835.0000
C00591=-47.575,-43.938,59.508,-179.6957,37.5811,-11837.2759
C00592=-49.608,-41.728,59.535,174.2083,36.7306,-11839.9310
C00593=-52.385,-39.754,60.163,160.9694,20.0893,-11842.8058
C00594=-55.279,-40.327,61.754,179.0540,0.1227,-11843.8886
C00595=-58.966,-42.664,63.969,-175.9921,-0.2034,-11844.1129
C00596=-63.647,-46.056,66.266,-173.7731,-0.1698,-11844.1099
C00597=-68.885,-49.892,68.033,-172.3610,-0.2408,-11844.0850
C00598=-73.964,-53.229,68.906,-172.5034,-1.7072,-11844.2589
C00599=-79.427,-53.903,69.366,-176.4883,-3.3136,-11845.8373
C00600=-84.528,-51.697,69.740,-179.1554,-2.2229,-11848.5502
C00601=-88.212,-47.022,70.117,-179.9990,-0.1564,-11851.9399
C00602=-91.079,-41.276,70.366,179.9981,-0.0180,-11855.6205
C00603=-93.589,-35.216,70.366,179.9993,-0.0181,-11859.3795
C00604=-95.625,-29.126,70.117,-179.9996,-0.1559,-11863.0600
C00605=-96.325,-23.215,69.740,179.1510,-2.2246,-11866.4497
C00606=-94.279,-18.048,69.366,176.4898,-3.3102,-11869.1629
C00607=-89.940,-14.662,68.906,172.5060,-1.7115,-11870.7411
C00608=-83.988,-13.430,68.033,172.3612,-0.2407,-11870.9151
C00609=-77.571,-12.439,66.266,173.7747,-0.1711,-11870.8898
C00610=-71.864,-11.527,63.969,175.9897,-0.1992,-11870.8874
C00611=-67.603,-10.572,61.754,-179.0583,0.1253,-11871.1119
C00612=-65.152,-8.932,60.163,-160.9703,20.0908,-11872.1937
C00613=-64.584,-5.572,59.535,-174.2146,36.7296,-11875.0690
C00614=-64.710,-2.572,59.508,179.6979,37.5837,-11877.7239
C00615=-64.758,0.000,59.526,-180.0000,37.5735,-11880.0000
C00616=-64.710,2.572,59.508,-179.6979,37.5837,-11882.2761
C00617=-64.584,5.572,59.535,174.2146,36.7296,-11884.9310
C00618=-65.152,8.932,60.163,160.9703,20.0908,-11887.8063
C00619=-67.603,10.572,61.754,179.0583,0.1253,-11888.8881
C00620=-71.864,11.527,63.969,-175.9897,-0.1992,-11889.1126
C00621=-77.571,12.439,66.266,-173.7747,-0.1711,-11889.1102
C00622=-83.988,13.430,68.033,-172.3612,-0.2407,-11889.0849
C00623=-89.940,14.662,68.906,-172.5060,-1.7115,-11889.2589
C00624=-94.279,18.048,69.366,-176.4898,-3.3102,-11890.8371
C00625=-96.325,23.215,69.740,-179.1510,-2.2246,-11893.5503
C00626=-95.625,29.126,70.117,179.9996,-0.1559,-11896.9400
C00627=-93.589,35.216,70.366,-179.9993,-0.0181,-11900.6205
C00628=-91.079,41.276,70.366,-179.9981,-0.0180,-11904.3795
C00629=-88.212,47.022,70.117,179.9990,-0.1564,-11908.0601
C00630=-84.528,51.697,69.740,179.1554,-2.2229,-11911.4498
C00631=-79.427,53.903,69.366,176.4883,-3.3136,-11914.1627
C00632=-73.964,53.229,68.906,172.5034,-1.7072,-11915.7411
C00633=-68.885,49.892,68.033,172.3610,-0.2408,-11915.9150
C00634=-63.647,46.056,66.266,173.7731,-0.1698,-11915.8901
C00635=-58.966,42.664,63.969,175.9921,-0.2034,-11915.8871
C00636=-55.279,40.327,61.754,-179.0540,0.1227,-11916.1114
C00637=-52.385,39.754,60.163,-160.9694,20.0893,-11917.1942
C00638=-49.608,41.728,59.535,-174.2183,36.7311,-11920.0690
C00639=-47.576,43.938,59.508,179.6961,37.5811,-11922.7235
C00640=-45.791,45.791,59.526,-180.0000,37.5739,-11925.0000
C00641=-43.938,47.575,59.508,-179.6957,37.5811,-11927.2759
C00642=-41.728,49.608,59.535,174.2083,36.7306,-11929.9310
C00643=-39.754,52.385,60.163,160.9694,20.0893,-11932.8058
C00644=-40.327,55.279,61.754,179.0540,0.1227,-11933.8886
C00645=-42.664,58.966,63.969,-175.9921,-0.2034,-11934.1129
C00646=-46.056,63.647,66.266,-173.7731,-0.1698,-11934.1099
C00647=-49.892,68.885,68.033,-172.3610,-0.2408,-11934.0850
C00648=-53.229,73.964,68.906,-172.5034,-1.7072,-11934.2589
C00649=-53.903,79.427,69.366,-176.4883,-3.3136,-11935.8373
C00650=-51.697,84.528,69.740,-179.1554,-2.2229,-11938.5502
C00651=-47.022,88.212,70.117,-179.9990,-0.1564,-11941.9399
C00652=-41.276,91.079,70.366,179.9981,-0.0180,-11945.6205
C00653=-35.216,93.589,70.366,179.9993,-0.0181,-11949.3795
C00654=-29.126,95.625,70.117,-179.9996,-0.1559,-11953.0600
C00655=-23.215,96.325,69.740,179.1510,-2.2246,-11956.4497
C00656=-18.048,94.279,69.366,176.4898,-3.3102,-11959.1629
C00657=-14.662,89.940,68.906,172.5060,-1.7115,-11960.7411
C00658=-13.430,83.988,68.033,172.3612,-0.2407,-11960.9151
C00659=-12.439,77.571,66.266,173.7747,-0.1711,-11960.8898
C00660=-11.527,71.864,63.969,175.9897,-0.1992,-11960.8874
C00661=-10.572,67.603,61.754,-179.0583,0.1253,-11961.1119
C00662=-8.932,65.152,60.163,-160.9703,20.0908,-11962.1937
C00663=-5.572,64.584,59.535,-174.2146,36.7296,-11965.0690
C00664=-2.572,64.710,59.508,179.6979,37.5837,-11967.7239
C00665=0.000,64.758,59.526,-180.0000,37.5735,-11970.0000
C00666=0.000,63.425,61.276,-180.0000,37.0005,-11970.0000
C00667=2.450,63.381,61.257,-179.6948,37.0092,-11972.2137
C00668=5.367,63.268,61.285,174.0310,36.0790,-11974.8488
C00669=8.682,63.886,61.945,161.4111,18.6823,-11977.7390
C00670=10.270,66.465,63.612,179.7526,0.0255,-11978.7837
C00671=11.189,70.924,65.929,-175.8210,-0.1771,-11978.9651
C00672=12.084,76.878,68.324,-173.8594,-0.1394,-11978.9329
C00673=13.063,83.550,70.157,-172.5965,-0.1926,-11978.8862
C00674=14.270,89.726,71.060,-172.7438,-1.5775,-11979.0366
C00675=17.683,94.235,71.535,-176.5649,-3.1765,-11980.6278
C00676=22.929,96.378,71.920,-179.1719,-2.1420,-11983.3823
C00677=28.946,95.684,72.309,-179.9969,-0.1487,-11986.8314
C00678=35.156,93.612,72.565,-179.9993,-0.0181,-11990.5837
C00679=41.335,91.053,72.565,-179.9981,-0.0180,-11994.4165
C00680=47.191,88.127,72.309,179.9965,-0.1513,-11998.1685
C00681=51.936,84.362,71.920,179.1729,-2.1445,-12001.6178
C00682=54.130,79.138,71.535,176.5613,-3.1804,-12004.3719
C00683=53.356,73.536,71.060,172.7432,-1.5739,-12005.9638
C00684=49.842,68.316,70.157,172.5980,-0.1884,-12006.1137
C00685=45.816,62.906,68.324,173.8645,-0.1373,-12006.0668
C00686=42.239,58.063,65.929,175.8220,-0.1746,-12006.0347
C00687=39.736,54.260,63.612,-179.7499,0.0269,-12006.2163
C00688=39.035,51.313,61.945,-161.4145,18.6787,-12007.2611
C00689=40.942,48.532,61.285,-174.0315,36.0780,-12010.1513
C00690=43.085,46.550,61.257,179.6995,37.0101,-12012.7862
C00691=44.848,44.848,61.276,-180.0000,36.9982,-12015.0000
C00692=46.550,43.085,61.257,-179.6995,37.0101,-12017.2138
C00693=48.532,40.942,61.285,174.0315,36.0780,-12019.8487
C00694=51.313,39.035,61.945,161.4145,18.6787,-12022.7389
C00695=54.260,39.736,63.612,179.7499,0.0269,-12023.7837
C00696=58.063,42.239,65.929,-175.8220,-0.1746,-12023.9653
C00697=62.906,45.816,68.324,-173.8645,-0.1373,-12023.9332
C00698=68.316,49.842,70.157,-172.5980,-0.1884,-12023.8863
C00699=73.536,53.356,71.060,-172.7432,-1.5739,-12024.0362
C00700=79.138,54.130,71.535,-176.5613,-3.1804,-12025.6281
C00701=84.362,51.936,71.920,-179.1729,-2.1445,-12028.3822
C00702=88.127,47.191,72.309,-179.9965,-0.1513,-12031.8315
C00703=91.053,41.335,72.565,179.9981,-0.0180,-12035.5835
C00704=93.612,35.156,72.565,179.9993,-0.0181,-12039.4163
C00705=95.684,28.946,72.309,179.9969,-0.1487,-12043.1686
C00706=96.378,22.929,71.920,179.1719,-2.1420,-12046.6177
C00707=94.235,17.683,71.535,176.5649,-3.1765,-12049.3722
C00708=89.726,14.270,71.060,172.7438,-1.5775,-12050.9634
C00709=83.550,13.063,70.157,172.5965,-0.1926,-12051.1138
C00710=76.878,12.084,68.324,173.8594,-0.1394,-12051.0671
C00711=70.924,11.189,65.929,175.8210,-0.1771,-12051.0349
C00712=66.465,10.270,63.612,-179.7526,0.0255,-12051.2163
C00713=63.886,8.682,61.945,-161.4111,18.6823,-12052.2610
C00714=63.268,5.367,61.285,-174.0310,36.0790,-12055.1512
C00715=63.381,2.450,61.257,179.6948,37.0092,-12057.7863
C00716=63.425,0.000,61.276,-180.0000,37.0005,-12060.0000
C00717=63.381,-2.450,61.257,-179.6948,37.0092,-12062.2137
C00718=63.268,-5.367,61.285,174.0310,36.0790,-12064.8488
C00719=63.886,-8.682,61.945,161.4119,18.6766,-12067.7390
C00720=66.465,-10.270,63.612,179.7526,0.0255,-12068.7837
C00721=70.924,-11.189,65.929,-175.8210,-0.1771,-12068.9651
C00722=76.878,-12.084,68.324,-173.8594,-0.1394,-12068.9329
C00723=83.550,-13.063,70.157,-172.5965,-0.1926,-12068.8862
C00724=89.726,-14.270,71.060,-172.7438,-1.5775,-12069.0366
C00725=94.235,-17.683,71.535,-176.5649,-3.1765,-12070.6278
C00726=96.378,-22.929,71.920,-179.1719,-2.1420,-12073.3823
C00727=95.684,-28.946,72.309,-179.9969,-0.1487,-12076.8314
C00728=93.612,-35.156,72.565,-179.9993,-0.0181,-12080.5837
C00729=91.053,-41.335,72.565,-179.9981,-0.0180,-12084.4165
C00730=88.127,-47.191,72.309,179.9965,-0.1513,-12088.1685
C00731=84.362,-51.936,71.920,179.1729,-2.1445,-12091.6178
C00732=79.138,-54.130,71.535,176.5613,-3.1804,-12094.3719
C00733=73.536,-53.356,71.060,172.7432,-1.5739,-12095.9638
C00734=68.316,-49.842,70.157,172.5980,-0.1884,-12096.1137
C00735=62.906,-45.816,68.324,173.8645,-0.1373,-12096.0668
C00736=58.063,-42.239,65.929,175.8220,-0.1746,-12096.0347
C00737=54.260,-39.736,63.612,-179.7499,0.0269,-12096.2163
C00738=51.313,-39.035,61.945,-161.4145,18.6787,-12097.2611
C00739=48.532,-40.942,61.285,-174.0315,36.0780,-12100.1513
C00740=46.550,-43.085,61.257,179.6995,37.0101,-12102.7862
C00741=44.848,-44.848,61.276,-180.0000,36.9982,-12105.0000
C00742=43.085,-46.550,61.257,-179.6995,37.0101,-12107.2138
C00743=40.942,-48.532,61.285,174.0315,36.0780,-12109.8487
C00744=39.035,-51.313,61.945,161.4145,18.6787,-12112.7389
C00745=39.736,-54.260,63.612,179.7499,0.0269,-12113.7837
C00746=42.239,-58.063,65.929,-175.8220,-0.1746,-12113.9653
C00747=45.816,-62.906,68.324,-173.8645,-0.1373,-12113.9332
C00748=49.842,-68.316,70.157,-172.5980,-0.1884,-12113.8863
C00749=53.356,-73.536,71.060,-172.7432,-1.5739,-12114.0362
C00750=54.130,-79.138,71.535,-176.5613,-3.1804,-12115.6281
C00751=51.936,-84.362,71.920,-179.1729,-2.1445,-12118.3822
C00752=47.191,-88.127,72.309,-179.9965,-0.1513,-12121.8315
C00753=41.335,-91.053,72.565,179.9981,-0.0180,-12125.5835
C00754=35.156,-93.612,72.565,179.9993,-0.0181,-12129.4163
C00755=28.946,-95.684,72.309,179.9969,-0.1487,-12133.1686
C00756=22.929,-96.378,71.920,179.1719,-2.1420,-12136.6177
C00757=17.683,-94.235,71.535,176.5649,-3.1765,-12139.3722
C00758=14.270,-89.726,71.060,172.7438,-1.5775,-12140.9634
C00759=13.063,-83.550,70.157,172.5965,-0.1926,-12141.1138
C00760=12.084,-76.878,68.324,173.8594,-0.1394,-12141.0671
C00761=11.189,-70.924,65.929,175.8210,-0.1771,-12141.0349
C00762=10.270,-66.465,63.612,-179.7526,0.0255,-12141.2163
C00763=8.682,-63.886,61.945,-161.4111,18.6823,-12142.2610
C00764=5.367,-63.268,61.285,-174.0310,36.0790,-12145.1512
C00765=2.450,-63.381,61.257,179.6948,37.0092,-12147.7863
C00766=0.000,-63.425,61.276,-180.0000,37.0005,-12150.0000
C00767=0.000,-63.425,61.276,-180.0000,37.0005,-12150.0000
C00768=-2.450,-63.381,61.257,-179.6948,37.0092,-12152.2137
C00769=-5.367,-63.268,61.285,174.0310,36.0790,-12154.8488
C00770=-8.682,-63.886,61.945,161.4119,18.6766,-12157.7390
C00771=-10.270,-66.465,63.612,179.7526,0.0255,-12158.7837
C00772=-11.189,-70.924,65.929,-175.8210,-0.1771,-12158.9651
C00773=-12.084,-76.878,68.324,-173.8594,-0.1394,-12158.9329
C00774=-13.063,-83.550,70.157,-172.5965,-0.1926,-12158.8862
C00775=-14.270,-89.726,71.060,-172.7438,-1.5775,-12159.0366
C00776=-17.683,-94.235,71.535,-176.5649,-3.1765,-12160.6278
C00777=-22.929,-96.378,71.920,-179.1719,-2.1420,-12163.3823
C00778=-28.946,-95.684,72.309,-179.9969,-0.1487,-12166.8314
C00779=-35.156,-93.612,72.565,-179.9993,-0.0181,-12170.5837
C00780=-41.335,-91.053,72.565,-179.9981,-0.0180,-12174.4165
C00781=-47.191,-88.127,72.309,179.9965,-0.1513,-12178.1685
C00782=-51.936,-84.362,71.920,179.1729,-2.1445,-12181.6178
C00783=-54.130,-79.138,71.535,176.5613,-3.1804,-12184.3719
C00784=-53.356,-73.536,71.060,172.7432,-1.5739,-12185.9638
C00785=-49.842,-68.316,70.157,172.5980,-0.1884,-12186.1137
C00786=-45.816,-62.906,68.324,173.8645,-0.1373,-12186.0668
C00787=-42.239,-58.063,65.929,175.8220,-0.1746,-12186.0347
C00788=-39.736,-54.260,63.612,-179.7499,0.0269,-12186.2163
C00789=-39.035,-51.313,61.945,-161.4145,18.6787,-12187.2611
C00790=-40.942,-48.532,61.285,-174.0315,36.0780,-12190.1513
C00791=-43.085,-46.550,61.257,179.6995,37.0101,-12192.7862
C00792=-44.848,-44.848,61.276,180.0000,36.9982,-12195.0000
C00793=-46.550,-43.085,61.257,-179.6995,37.0101,-12197.2138
C00794=-48.532,-40.942,61.285,174.0315,36.0780,-12199.8487
C00795=-51.313,-39.035,61.945,161.4145,18.6787,-12202.7389
C00796=-54.260,-39.736,63.612,179.7499,0.0269,-12203.7837
C00797=-58.063,-42.239,65.929,-175.8220,-0.1746,-12203.9653
C00798=-62.906,-45.816,68.324,-173.8645,-0.1373,-12203.9332
C00799=-68.316,-49.842,70.157,-172.5980,-0.1884,-12203.8863
C00800=-73.536,-53.356,71.060,-172.7432,-1.5739,-12204.0362
C00801=-79.138,-54.130,71.535,-176.5613,-3.1804,-12205.6281
C00802=-84.362,-51.936,71.920,-179.1729,-2.1445,-12208.3822
C00803=-88.127,-47.191,72.309,-179.9965,-0.1513,-12211.8315
C00804=-91.053,-41.335,72.565,179.9981,-0.0180,-12215.5835
C00805=-93.612,-35.156,72.565,179.9993,-0.0181,-12219.4163
C00806=-95.684,-28.946,72.309,179.9969,-0.1487,-12223.1686
C00807=-96.378,-22.929,71.920,179.1719,-2.1420,-12226.6177
C00808=-94.235,-17.683,71.535,176.5649,-3.1765,-12229.3722
C00809=-89.726,-14.270,71.060,172.7438,-1.5775,-12230.9634
C00810=-83.550,-13.063,70.157,172.5965,-0.1926,-12231.1138
C00811=-76.878,-12.084,68.324,173.8594,-0.1394,-12231.0671
C00812=-70.924,-11.189,65.929,175.8210,-0.1771,-12231.0349
C00813=-66.465,-10.270,63.612,-179.7526,0.0255,-12231.2163
C00814=-63.886,-8.682,61.945,-161.4111,18.6823,-12232.2610
C00815=-63.268,-5.367,61.285,-174.0310,36.0790,-12235.1512
C00816=-63.381,-2.450,61.257,179.6948,37.0092,-12237.7863
C00817=-63.425,0.000,61.276,180.0000,37.0005,-12240.0000
C00818=-63.381,2.450,61.257,-179.6948,37.0092,-12242.2137
C00819=-63.268,5.367,61.285,174.0310,36.0790,-12244.8488
C00820=-63.886,8.682,61.945,161.4119,18.6766,-12247.7390
C00821=-66.465,10.270,63.612,179.7526,0.0255,-12248.7837
C00822=-70.924,11.189,65.929,-175.8210,-0.1771,-12248.9651
C00823=-76.878,12.084,68.324,-173.8594,-0.1394,-12248.9329
C00824=-83.550,13.063,70.157,-172.5965,-0.1926,-12248.8862
C00825=-89.726,14.270,71.060,-172.7438,-1.5775,-12249.0366
C00826=-94.235,17.683,71.535,-176.5649,-3.1765,-12250.6278
C00827=-96.378,22.929,71.920,-179.1719,-2.1420,-12253.3823
C00828=-95.684,28.946,72.309,-179.9969,-0.1487,-12256.8314
C00829=-93.612,35.156,72.565,-179.9993,-0.0181,-12260.5837
C00830=-91.053,41.335,72.565,-179.9981,-0.0180,-12264.4165
C00831=-88.127,47.191,72.309,179.9965,-0.1513,-12268.1685
C00832=-84.362,51.936,71.920,179.1729,-2.1445,-12271.6178
C00833=-79.138,54.130,71.535,176.5613,-3.1804,-12274.3719
C00834=-73.536,53.356,71.060,172.7432,-1.5739,-12275.9638
C00835=-68.316,49.842,70.157,172.5980,-0.1884,-12276.1137
C00836=-62.906,45.816,68.324,173.8645,-0.1373,-12276.0668
C00837=-58.063,42.239,65.929,175.8220,-0.1746,-12276.0347
C00838=-54.260,39.736,63.612,-179.7499,0.0269,-12276.2163
C00839=-51.313,39.035,61.945,-161.4145,18.6787,-12277.2611
C00840=-48.532,40.942,61.285,-174.0315,36.0780,-12280.1513
C00841=-46.550,43.085,61.257,179.6995,37.0101,-12282.7862
C00842=-44.848,44.848,61.276,180.0000,36.9982,-12285.0000
C00843=-43.085,46.550,61.257,-179.6995,37.0101,-12287.2138
C00844=-40.942,48.532,61.285,174.0315,36.0780,-12289.8487
C00845=-39.035,51.313,61.945,161.4145,18.6787,-12292.7389
C00846=-39.736,54.260,63.612,179.7499,0.0269,-12293.7837
C00847=-42.239,58.063,65.929,-175.8220,-0.1746,-12293.9653
C00848=-45.816,62.906,68.324,-173.8645,-0.1373,-12293.9332
C00849=-49.842,68.316,70.157,-172.5980,-0.1884,-12293.8863
C00850=-53.356,73.536,71.060,-172.7432,-1.5739,-12294.0362
C00851=-54.130,79.138,71.535,-176.5613,-3.1804,-12295.6281
C00852=-51.936,84.362,71.920,-179.1729,-2.1445,-12298.3822
C00853=-47.191,88.127,72.309,-179.9965,-0.1513,-12301.8315
C00854=-41.335,91.053,72.565,179.9981,-0.0180,-12305.5835
C00855=-35.156,93.612,72.565,179.9993,-0.0181,-12309.4163
C00856=-28.946,95.684,72.309,179.9969,-0.1487,-12313.1686
C00857=-22.929,96.378,71.920,179.1719,-2.1420,-12316.6177
C00858=-17.683,94.235,71.535,176.5649,-3.1765,-12319.3722
C00859=-14.270,89.726,71.060,172.7438,-1.5775,-12320.9634
C00860=-13.063,83.550,70.157,172.5965,-0.1926,-12321.1138
C00861=-12.084,76.878,68.324,173.8594,-0.1394,-12321.0671
C00862=-11.189,70.924,65.929,175.8210,-0.1771,-12321.0349
C00863=-10.270,66.465,63.612,-179.7526,0.0255,-12321.2163
C00864=-8.682,63.886,61.945,-161.4119,18.6766,-12322.2610
C00865=-5.367,63.268,61.285,-174.0310,36.0790,-12325.1512
C00866=-2.450,63.381,61.257,179.6948,37.0092,-12327.7863
C00867=0.000,63.425,61.276,180.0000,37.0005,-12330.0000
C00868=0.000,62.111,63.041,180.0000,36.3256,-12330.0000
C00869=2.330,62.072,63.021,-179.7028,36.3324,-12332.1497
C00870=5.165,61.970,63.050,173.8802,35.3262,-12334.7644
C00871=8.436,62.639,63.741,161.9639,17.2722,-12337.6702
C00872=9.975,65.350,65.485,-179.6415,-0.0322,-12338.6786
C00873=10.861,70.011,67.904,-175.7229,-0.1493,-12338.8182
C00874=11.743,76.212,70.393,-174.0066,-0.1107,-12338.7594
C00875=12.712,83.133,72.289,-172.8940,-0.1461,-12338.6938
C00876=13.898,89.524,73.219,-173.0501,-1.4397,-12338.8243
C00877=17.338,94.193,73.707,-176.6773,-3.0198,-12340.4296
C00878=22.659,96.427,74.103,-179.2016,-2.0437,-12343.2238
C00879=28.778,95.739,74.502,-179.9988,-0.1432,-12346.7302
C00880=35.099,93.634,74.765,-179.9993,-0.0181,-12350.5487
C00881=41.391,91.028,74.765,-179.9981,-0.0180,-12354.4516
C00882=47.349,88.047,74.502,179.9991,-0.1436,-12358.2700
C00883=52.162,84.206,74.103,179.2030,-2.0441,-12361.7764
C00884=54.344,78.865,73.707,176.6784,-3.0215,-12364.5698
C00885=53.475,73.130,73.219,173.0551,-1.4407,-12366.1755
C00886=49.795,67.773,72.289,172.8935,-0.1468,-12366.3059
C00887=45.586,62.194,70.393,174.0079,-0.1079,-12366.2401
C00888=41.825,57.185,67.904,175.7207,-0.1531,-12366.1817
C00889=39.156,53.262,65.485,179.6421,-0.0355,-12366.3218
C00890=38.328,50.258,63.741,-161.9596,17.2759,-12367.3300
C00891=40.167,47.472,63.050,-173.8825,35.3269,-12370.2352
C00892=42.244,45.539,63.021,179.7046,36.3332,-12372.8504
C00893=43.919,43.919,63.041,-180.0000,36.3263,-12375.0000
C00894=45.539,42.244,63.021,-179.7046,36.3332,-12377.1496
C00895=47.472,40.167,63.050,173.8780,35.3233,-12379.7648
C00896=50.258,38.328,63.741,161.9596,17.2759,-12382.6700
C00897=53.262,39.156,65.485,-179.6421,-0.0355,-12383.6782
C00898=57.185,41.825,67.904,-175.7207,-0.1531,-12383.8183
C00899=62.194,45.586,70.393,-174.0079,-0.1079,-12383.7599
C00900=67.773,49.795,72.289,-172.8935,-0.1468,-12383.6941
C00901=73.130,53.475,73.219,-173.0551,-1.4407,-12383.8245
C00902=78.865,54.344,73.707,-176.6784,-3.0215,-12385.4302
C00903=84.206,52.162,74.103,-179.2030,-2.0441,-12388.2236
C00904=88.047,47.349,74.502,-179.9991,-0.1436,-12391.7300
C00905=91.028,41.391,74.765,179.9981,-0.0180,-12395.5484
C00906=93.634,35.099,74.765,179.9993,-0.0181,-12399.4513
C00907=95.739,28.778,74.502,179.9988,-0.1432,-12403.2698
C00908=96.427,22.659,74.103,179.2016,-2.0437,-12406.7762
C00909=94.193,17.338,73.707,176.6773,-3.0198,-12409.5704
C00910=89.524,13.898,73.219,173.0501,-1.4397,-12411.1757
C00911=83.133,12.712,72.289,172.8940,-0.1461,-12411.3062
C00912=76.212,11.743,70.393,174.0066,-0.1107,-12411.2406
C00913=70.011,10.861,67.904,175.7229,-0.1493,-12411.1818
C00914=65.350,9.975,65.485,179.6415,-0.0322,-12411.3214
C00915=62.639,8.436,63.741,-161.9639,17.2722,-12412.3298
C00916=61.970,5.165,63.050,-173.8802,35.3262,-12415.2356
C00917=62.072,2.330,63.021,179.7028,36.3324,-12417.8503
C00918=62.111,0.000,63.041,-180.0000,36.3256,-12420.0000
C00919=62.072,-2.330,63.021,-179.7028,36.3324,-12422.1497
C00920=61.970,-5.165,63.050,173.8802,35.3262,-12424.7644
C00921=62.640,-8.436,63.741,161.9639,17.2723,-12427.6701
C00922=65.350,-9.975,65.485,-179.6415,-0.0322,-12428.6786
C00923=70.011,-10.861,67.904,-175.7229,-0.1493,-12428.8182
C00924=76.212,-11.743,70.393,-174.0066,-0.1107,-12428.7594
C00925=83.133,-12.712,72.289,-172.8940,-0.1461,-12428.6938
C00926=89.524,-13.898,73.219,-173.0501,-1.4397,-12428.8243
C00927=94.193,-17.338,73.707,-176.6773,-3.0198,-12430.4296
C00928=96.427,-22.659,74.103,-179.2016,-2.0437,-12433.2238
C00929=95.739,-28.778,74.502,-179.9988,-0.1432,-12436.7302
C00930=93.634,-35.099,74.765,-179.9993,-0.0181,-12440.5487
C00931=91.028,-41.391,74.765,-179.9981,-0.0180,-12444.4516
C00932=88.047,-47.349,74.502,179.9991,-0.1436,-12448.2700
C00933=84.206,-52.162,74.103,179.2030,-2.0441,-12451.7764
C00934=78.865,-54.344,73.707,176.6784,-3.0215,-12454.5698
C00935=73.130,-53.475,73.219,173.0551,-1.4407,-12456.1755
C00936=67.773,-49.795,72.289,172.8935,-0.1468,-12456.3059
C00937=62.194,-45.586,70.393,174.0079,-0.1079,-12456.2401
C00938=57.185,-41.825,67.904,175.7207,-0.1531,-12456.1817
C00939=53.262,-39.156,65.485,179.6421,-0.0355,-12456.3218
C00940=50.258,-38.328,63.741,-161.9596,17.2759,-12457.3300
C00941=47.472,-40.167,63.050,-173.8825,35.3269,-12460.2352
C00942=45.539,-42.244,63.021,179.7046,36.3332,-12462.8504
C00943=43.919,-43.919,63.041,-180.0000,36.3263,-12465.0000
C00944=42.244,-45.539,63.021,-179.7046,36.3332,-12467.1496
C00945=40.167,-47.472,63.050,173.8780,35.3233,-12469.7648
C00946=38.328,-50.258,63.741,161.9596,17.2759,-12472.6700
C00947=39.156,-53.262,65.485,-179.6421,-0.0355,-12473.6782
C00948=41.825,-57.185,67.904,-175.7207,-0.1531,-12473.8183
C00949=45.586,-62.194,70.393,-174.0079,-0.1079,-12473.7599
C00950=49.795,-67.773,72.289,-172.8935,-0.1468,-12473.6941
C00951=53.475,-73.130,73.219,-173.0551,-1.4407,-12473.8245
C00952=54.344,-78.865,73.707,-176.6784,-3.0215,-12475.4302
C00953=52.162,-84.206,74.103,-179.2030,-2.0441,-12478.2236
C00954=47.349,-88.047,74.502,-179.9991,-0.1436,-12481.7300
C00955=41.391,-91.028,74.765,179.9981,-0.0180,-12485.5484
C00956=35.099,-93.634,74.765,179.9993,-0.0181,-12489.4513
C00957=28.778,-95.739,74.502,179.9988,-0.1432,-12493.2698
C00958=22.659,-96.427,74.103,179.2016,-2.0437,-12496.7762
C00959=17.338,-94.193,73.707,176.6773,-3.0198,-12499.5704
C00960=13.898,-89.524,73.219,173.0501,-1.4397,-12501.1757
C00961=12.712,-83.133,72.289,172.8940,-0.1461,-12501.3062
C00962=11.743,-76.212,70.393,174.0066,-0.1107,-12501.2406
C00963=10.861,-70.011,67.904,175.7229,-0.1493,-12501.1818
C00964=9.975,-65.350,65.485,179.6415,-0.0322,-12501.3214
C00965=8.436,-62.639,63.741,-161.9639,17.2722,-12502.3298
C00966=5.165,-61.970,63.050,-173.8802,35.3262,-12505.2356
C00967=2.330,-62.072,63.021,179.7028,36.3324,-12507.8503
C00968=0.000,-62.111,63.041,-180.0000,36.3256,-12510.0000
C00969=0.000,-62.111,63.041,-180.0000,36.3256,-12510.0000
C00970=-2.330,-62.072,63.021,-179.7028,36.3324,-12512.1497
C00971=-5.165,-61.970,63.050,173.8802,35.3262,-12514.7644
C00972=-8.436,-62.640,63.741,161.9639,17.2723,-12517.6701
C00973=-9.975,-65.350,65.485,-179.6415,-0.0322,-12518.6786
C00974=-10.861,-70.011,67.904,-175.7229,-0.1493,-12518.8182
C00975=-11.743,-76.212,70.393,-174.0066,-0.1107,-12518.7594
C00976=-12.712,-83.133,72.289,-172.8940,-0.1461,-12518.6938
C00977=-13.898,-89.524,73.219,-173.0501,-1.4397,-12518.8243
C00978=-17.338,-94.193,73.707,-176.6773,-3.0198,-12520.4296
C00979=-22.659,-96.427,74.103,-179.2016,-2.0437,-12523.2238
C00980=-28.778,-95.739,74.502,-179.9988,-0.1432,-12526.7302
C00981=-35.099,-93.634,74.765,-179.9993,-0.0181,-12530.5487
C00982=-41.391,-91.028,74.765,-179.9981,-0.0180,-12534.4516
C00983=-47.349,-88.047,74.502,179.9991,-0.1436,-12538.2700
C00984=-52.162,-84.206,74.103,179.2030,-2.0441,-12541.7764
C00985=-54.344,-78.865,73.707,176.6784,-3.0215,-12544.5698
C00986=-53.475,-73.130,73.219,173.0551,-1.4407,-12546.1755
C00987=-49.795,-67.773,72.289,172.8935,-0.1468,-12546.3059
C00988=-45.586,-62.194,70.393,174.0079,-0.1079,-12546.2401
C00989=-41.825,-57.185,67.904,175.7207,-0.1531,-12546.1817
C00990=-39.156,-53.262,65.485,179.6421,-0.0355,-12546.3218
C00991=-38.328,-50.258,63.741,-161.9596,17.2759,-12547.3300
C00992=-40.167,-47.472,63.050,-173.8825,35.3269,-12550.2352
C00993=-42.244,-45.539,63.021,179.7046,36.3332,-12552.8504
C00994=-43.919,-43.919,63.041,-180.0000,36.3263,-12555.0000
C00995=-45.539,-42.244,63.021,-179.7046,36.3332,-12557.1496
C00996=-47.472,-40.167,63.050,173.8780,35.3233,-12559.7648
C00997=-50.258,-38.328,63.741,161.9596,17.2759,-12562.6700
C00998=-53.262,-39.156,65.485,-179.6421,-0.0355,-12563.6782
C00999=-57.185,-41.825,67.904,-175.7207,-0.1531,-12563.8183
C01000=-62.194,-45.586,70.393,-174.0079,-0.1079,-12563.7599
C01001=-67.773,-49.795,72.289,-172.8935,-0.1468,-12563.6941
C01002=-73.130,-53.475,73.219,-173.0551,-1.4407,-12563.8245
C01003=-78.865,-54.344,73.707,-176.6784,-3.0215,-12565.4302
C01004=-84.206,-52.162,74.103,-179.2030,-2.0441,-12568.2236
C01005=-88.047,-47.349,74.502,-179.9991,-0.1436,-12571.7300
C01006=-91.028,-41.391,74.765,179.9981,-0.0180,-12575.5484
C01007=-93.634,-35.099,74.765,179.9993,-0.0181,-12579.4513
C01008=-95.739,-28.778,74.502,179.9988,-0.1432,-12583.2698
C01009=-96.427,-22.659,74.103,179.2016,-2.0437,-12586.7762
C01010=-94.193,-17.338,73.707,176.6773,-3.0198,-12589.5704
C01011=-89.524,-13.898,73.219,173.0501,-1.4397,-12591.1757
C01012=-83.133,-12.712,72.289,172.8940,-0.1461,-12591.3062
C01013=-76.212,-11.743,70.393,174.0066,-0.1107,-12591.2406
C01014=-70.011,-10.861,67.904,175.7229,-0.1493,-12591.1818
C01015=-65.350,-9.975,65.485,179.6415,-0.0322,-12591.3214
C01016=-62.639,-8.436,63.741,-161.9639,17.2722,-12592.3298
C01017=-61.970,-5.165,63.050,-173.8802,35.3262,-12595.2356
C01018=-62.072,-2.330,63.021,179.7028,36.3324,-12597.8503
C01019=-62.111,0.000,63.041,-180.0000,36.3256,-12600.0000
C01020=-62.072,2.330,63.021,-179.7028,36.3324,-12602.1497
C01021=-61.970,5.165,63.050,173.8802,35.3262,-12604.7644
C01022=-62.640,8.436,63.741,161.9639,17.2723,-12607.6701
C01023=-65.350,9.975,65.485,-179.6415,-0.0322,-12608.6786
C01024=-70.011,10.861,67.904,-175.7229,-0.1493,-12608.8182
C01025=-76.212,11.743,70.393,-174.0066,-0.1107,-12608.7594
C01026=-83.133,12.712,72.289,-172.8940,-0.1461,-12608.6938
C01027=-89.524,13.898,73.219,-173.0501,-1.4397,-12608.8243
C01028=-94.193,17.338,73.707,-176.6773,-3.0198,-12610.4296
C01029=-96.427,22.659,74.103,-179.2016,-2.0437,-12613.2238
C01030=-95.739,28.778,74.502,-179.9988,-0.1432,-12616.7302
C01031=-93.634,35.099,74.765,-179.9993,-0.0181,-12620.5487
C01032=-91.028,41.391,74.765,-179.9981,-0.0180,-12624.4516
C01033=-88.047,47.349,74.502,179.9991,-0.1436,-12628.2700
C01034=-84.206,52.162,74.103,179.2030,-2.0441,-12631.7764
C01035=-78.865,54.344,73.707,176.6784,-3.0215,-12634.5698
C01036=-73.130,53.475,73.219,173.0551,-1.4407,-12636.1755
C01037=-67.773,49.795,72.289,172.8935,-0.1468,-12636.3059
C01038=-62.194,45.586,70.393,174.0079,-0.1079,-12636.2401
C01039=-57.185,41.825,67.904,175.7207,-0.1531,-12636.1817
C01040=-53.262,39.156,65.485,179.6421,-0.0355,-12636.3218
C01041=-50.258,38.328,63.741,-161.9596,17.2759,-12637.3300
C01042=-47.472,40.167,63.050,-173.8825,35.3269,-12640.2352
C01043=-45.539,42.244,63.021,179.7046,36.3332,-12642.8504
C01044=-43.919,43.919,63.041,180.0000,36.3263,-12645.0000
C01045=-42.244,45.539,63.021,-179.7046,36.3332,-12647.1496
C01046=-40.167,47.472,63.050,173.8780,35.3233,-12649.7648
C01047=-38.328,50.258,63.741,161.9596,17.2759,-12652.6700
C01048=-39.156,53.262,65.485,-179.6421,-0.0355,-12653.6782
C01049=-41.825,57.185,67.904,-175.7207,-0.1531,-12653.8183
C01050=-45.586,62.194,70.393,-174.0079,-0.1079,-12653.7599
C01051=-49.795,67.773,72.289,-172.8935,-0.1468,-12653.6941
C01052=-53.475,73.130,73.219,-173.0551,-1.4407,-12653.8245
C01053=-54.344,78.865,73.707,-176.6784,-3.0215,-12655.4302
C01054=-52.162,84.206,74.103,-179.2030,-2.0441,-12658.2236
C01055=-47.349,88.047,74.502,-179.9991,-0.1436,-12661.7300
C01056=-41.391,91.028,74.765,179.9981,-0.0180,-12665.5484
C01057=-35.099,93.634,74.765,179.9993,-0.0181,-12669.4513
C01058=-28.778,95.739,74.502,179.9988,-0.1432,-12673.2698
C01059=-22.659,96.427,74.103,179.2016,-2.0437,-12676.7762
C01060=-17.338,94.193,73.707,176.6773,-3.0198,-12679.5704
C01061=-13.898,89.524,73.219,173.0501,-1.4397,-12681.1757
C01062=-12.712,83.133,72.289,172.8940,-0.1461,-12681.3062
C01063=-11.743,76.212,70.393,174.0066,-0.1107,-12681.2406
C01064=-10.861,70.011,67.904,175.7229,-0.1493,-12681.1818
C01065=-9.975,65.350,65.485,179.6415,-0.0322,-12681.3214
C01066=-8.436,62.640,63.741,-161.9639,17.2723,-12682.3299
C01067=-5.165,61.970,63.050,-173.8802,35.3262,-12685.2356
C01068=-2.330,62.072,63.021,179.7028,36.3324,-12687.8503
C01069=0.000,62.111,63.041,180.0000,36.3256,-12690.0000
C01070=0.000,60.820,64.822,180.0000,35.5497,-12690.0000
C01071=2.212,60.785,64.801,-179.7074,35.5593,-12692.0841
C01072=4.967,60.695,64.832,173.7605,34.4682,-12694.6784
C01073=8.195,61.417,65.554,162.6105,15.8904,-12697.6002
C01074=9.686,64.262,67.375,-179.1259,-0.0711,-12698.5715
C01075=10.544,69.129,69.894,-175.6880,-0.1257,-12698.6723
C01076=11.418,75.576,72.474,-174.2120,-0.0836,-12698.5913
C01077=12.382,82.740,74.428,-173.2591,-0.1124,-12698.5111
C01078=13.550,89.334,75.383,-173.4296,-1.3094,-12698.6248
C01079=17.016,94.154,75.883,-176.8342,-2.8344,-12700.2442
C01080=22.407,96.473,76.288,-179.2397,-1.9299,-12703.0758
C01081=28.621,95.791,76.696,179.9993,-0.1377,-12706.6354
C01082=35.046,93.654,76.964,-179.9993,-0.0181,-12710.5162
C01083=41.442,91.005,76.964,-179.9981,-0.0180,-12714.4836
C01084=47.497,87.973,76.696,-179.9983,-0.1358,-12718.3648
C01085=52.372,84.060,76.288,179.2407,-1.9248,-12721.9242
C01086=54.545,78.609,75.883,176.8367,-2.8312,-12724.7559
C01087=53.588,72.750,75.383,173.4272,-1.3089,-12726.3755
C01088=49.751,67.261,74.428,173.2583,-0.1085,-12726.4893
C01089=45.367,61.514,72.474,174.2127,-0.0823,-12726.4090
C01090=41.426,56.337,69.894,175.6860,-0.1257,-12726.3280
C01091=38.591,52.289,67.375,179.1285,-0.0735,-12726.4285
C01092=37.634,49.223,65.554,-162.6128,15.8893,-12727.4001
C01093=39.406,46.429,64.832,-173.7617,34.4707,-12730.3225
C01094=41.417,44.545,64.801,179.7113,35.5606,-12732.9160
C01095=43.006,43.006,64.822,180.0000,35.5489,-12735.0000
C01096=44.545,41.417,64.801,-179.7113,35.5606,-12737.0840
C01097=46.430,39.405,64.832,173.7564,34.4670,-12739.6788
C01098=49.223,37.634,65.554,162.6128,15.8893,-12742.5999
C01099=52.289,38.591,67.375,-179.1285,-0.0735,-12743.5715
C01100=56.337,41.426,69.894,-175.6860,-0.1257,-12743.6720
C01101=61.514,45.367,72.474,-174.2127,-0.0823,-12743.5910
C01102=67.261,49.751,74.428,-173.2583,-0.1085,-12743.5107
C01103=72.750,53.588,75.383,-173.4272,-1.3089,-12743.6245
C01104=78.609,54.545,75.883,-176.8367,-2.8312,-12745.2441
C01105=84.060,52.372,76.288,-179.2407,-1.9248,-12748.0758
C01106=87.973,47.497,76.696,179.9983,-0.1358,-12751.6352
C01107=91.005,41.442,76.964,179.9981,-0.0180,-12755.5164
C01108=93.654,35.046,76.964,179.9993,-0.0181,-12759.4838
C01109=95.791,28.621,76.696,-179.9993,-0.1377,-12763.3646
C01110=96.473,22.407,76.288,179.2397,-1.9299,-12766.9242
C01111=94.154,17.016,75.883,176.8342,-2.8344,-12769.7558
C01112=89.334,13.550,75.383,173.4296,-1.3094,-12771.3752
C01113=82.740,12.382,74.428,173.2591,-0.1124,-12771.4889
C01114=75.576,11.418,72.474,174.2120,-0.0836,-12771.4087
C01115=69.129,10.544,69.894,175.6880,-0.1257,-12771.3277
C01116=64.262,9.686,67.375,179.1259,-0.0711,-12771.4285
C01117=61.417,8.195,65.554,-162.6105,15.8904,-12772.3998
C01118=60.695,4.967,64.832,-173.7605,34.4682,-12775.3216
C01119=60.785,2.212,64.801,179.7074,35.5593,-12777.9159
C01120=60.820,0.000,64.822,180.0000,35.5497,-12780.0000
C01121=60.785,-2.212,64.801,-179.7074,35.5593,-12782.0841
C01122=60.695,-4.967,64.832,173.7605,34.4682,-12784.6784
C01123=61.417,-8.195,65.554,162.6105,15.8904,-12787.6002
C01124=64.262,-9.686,67.375,-179.1259,-0.0711,-12788.5715
C01125=69.129,-10.544,69.894,-175.6880,-0.1257,-12788.6723
C01126=75.576,-11.418,72.474,-174.2120,-0.0836,-12788.5913
C01127=82.740,-12.382,74.428,-173.2591,-0.1124,-12788.5111
C01128=89.334,-13.550,75.383,-173.4296,-1.3094,-12788.6248
C01129=94.154,-17.016,75.883,-176.8342,-2.8344,-12790.2442
C01130=96.473,-22.407,76.288,-179.2397,-1.9299,-12793.0758
C01131=95.791,-28.621,76.696,179.9993,-0.1377,-12796.6354
C01132=93.654,-35.046,76.964,-179.9993,-0.0181,-12800.5162
C01133=91.005,-41.442,76.964,-179.9981,-0.0180,-12804.4836
C01134=87.973,-47.497,76.696,-179.9983,-0.1358,-12808.3648
C01135=84.060,-52.372,76.288,179.2407,-1.9248,-12811.9242
C01136=78.609,-54.545,75.883,176.8367,-2.8312,-12814.7559
C01137=72.750,-53.588,75.383,173.4272,-1.3089,-12816.3755
C01138=67.261,-49.751,74.428,173.2583,-0.1085,-12816.4893
C01139=61.514,-45.367,72.474,174.2127,-0.0823,-12816.4090
C01140=56.337,-41.426,69.894,175.6860,-0.1257,-12816.3280
C01141=52.289,-38.591,67.375,179.1285,-0.0735,-12816.4285
C01142=49.223,-37.634,65.554,-162.6128,15.8893,-12817.4001
C01143=46.429,-39.406,64.832,-173.7617,34.4707,-12820.3225
C01144=44.545,-41.417,64.801,179.7113,35.5606,-12822.9160
C01145=43.006,-43.006,64.822,-180.0000,35.5489,-12825.0000
C01146=41.417,-44.545,64.801,-179.7113,35.5606,-12827.0840
C01147=39.405,-46.430,64.832,173.7564,34.4670,-12829.6788
C01148=37.634,-49.223,65.554,162.6128,15.8893,-12832.5999
C01149=38.591,-52.289,67.375,-179.1285,-0.0735,-12833.5715
C01150=41.426,-56.337,69.894,-175.6860,-0.1257,-12833.6720
C01151=45.367,-61.514,72.474,-174.2127,-0.0823,-12833.5910
C01152=49.751,-67.261,74.428,-173.2583,-0.1085,-12833.5107
C01153=53.588,-72.750,75.383,-173.4272,-1.3089,-12833.6245
C01154=54.545,-78.609,75.883,-176.8367,-2.8312,-12835.2441
C01155=52.372,-84.060,76.288,-179.2407,-1.9248,-12838.0758
C01156=47.497,-87.973,76.696,179.9983,-0.1358,-12841.6352
C01157=41.442,-91.005,76.964,179.9981,-0.0180,-12845.5164
C01158=35.046,-93.654,76.964,179.9993,-0.0181,-12849.4838
C01159=28.621,-95.791,76.696,-179.9993,-0.1377,-12853.3646
C01160=22.407,-96.473,76.288,179.2397,-1.9299,-12856.9242
C01161=17.016,-94.154,75.883,176.8342,-2.8344,-12859.7558
C01162=13.550,-89.334,75.383,173.4296,-1.3094,-12861.3752
C01163=12.382,-82.740,74.428,173.2591,-0.1124,-12861.4889
C01164=11.418,-75.576,72.474,174.2120,-0.0836,-12861.4087
C01165=10.544,-69.129,69.894,175.6880,-0.1257,-12861.3277
C01166=9.686,-64.262,67.375,179.1259,-0.0711,-12861.4285
C01167=8.195,-61.417,65.554,-162.6105,15.8904,-12862.3998
C01168=4.967,-60.695,64.832,-173.7605,34.4682,-12865.3216
C01169=2.212,-60.785,64.801,179.7074,35.5593,-12867.9159
C01170=0.000,-60.820,64.822,-180.0000,35.5497,-12870.0000
C01171=0.000,-60.820,64.822,-180.0000,35.5497,-12870.0000
C01172=-2.212,-60.785,64.801,-179.7074,35.5593,-12872.0841
C01173=-4.967,-60.695,64.832,173.7605,34.4682,-12874.6784
C01174=-8.195,-61.417,65.554,162.6105,15.8904,-12877.6002
C01175=-9.686,-64.262,67.375,-179.1259,-0.0711,-12878.5715
C01176=-10.544,-69.129,69.894,-175.6880,-0.1257,-12878.6723
C01177=-11.418,-75.576,72.474,-174.2120,-0.0836,-12878.5913
C01178=-12.382,-82.740,74.428,-173.2591,-0.1124,-12878.5111
C01179=-13.550,-89.334,75.383,-173.4296,-1.3094,-12878.6248
C01180=-17.016,-94.154,75.883,-176.8342,-2.8344,-12880.2442
C01181=-22.407,-96.473,76.288,-179.2397,-1.9299,-12883.0758
C01182=-28.621,-95.791,76.696,179.9993,-0.1377,-12886.6354
C01183=-35.046,-93.654,76.964,-179.9993,-0.0181,-12890.5162
C01184=-41.442,-91.005,76.964,-179.9981,-0.0180,-12894.4836
C01185=-47.497,-87.973,76.696,-179.9983,-0.1358,-12898.3648
C01186=-52.372,-84.060,76.288,179.2407,-1.9248,-12901.9242
C01187=-54.545,-78.609,75.883,176.8367,-2.8312,-12904.7559
C01188=-53.588,-72.750,75.383,173.4272,-1.3089,-12906.3755
C01189=-49.751,-67.261,74.428,173.2583,-0.1085,-12906.4893
C01190=-45.367,-61.514,72.474,174.2127,-0.0823,-12906.4090
C01191=-41.426,-56.337,69.894,175.6860,-0.1257,-12906.3280
C01192=-38.591,-52.289,67.375,179.1285,-0.0735,-12906.4285
C01193=-37.634,-49.223,65.554,-162.6128,15.8893,-12907.4001
C01194=-39.406,-46.429,64.832,-173.7617,34.4707,-12910.3225
C01195=-41.417,-44.545,64.801,179.7113,35.5606,-12912.9160
C01196=-43.006,-43.006,64.822,-180.0000,35.5489,-12915.0000
C01197=-44.545,-41.417,64.801,-179.7113,35.5606,-12917.0840
C01198=-46.430,-39.405,64.832,173.7564,34.4670,-12919.6788
C01199=-49.223,-37.634,65.554,162.6128,15.8893,-12922.5999
C01200=-52.289,-38.591,67.375,-179.1285,-0.0735,-12923.5715
C01201=-56.337,-41.426,69.894,-175.6860,-0.1257,-12923.6720
C01202=-61.514,-45.367,72.474,-174.2127,-0.0823,-12923.5910
C01203=-67.261,-49.751,74.428,-173.2583,-0.1085,-12923.5107
C01204=-72.750,-53.588,75.383,-173.4272,-1.3089,-12923.6245
C01205=-78.609,-54.545,75.883,-176.8367,-2.8312,-12925.2441
C01206=-84.060,-52.372,76.288,-179.2407,-1.9248,-12928.0758
C01207=-87.973,-47.497,76.696,179.9983,-0.1358,-12931.6352
C01208=-91.005,-41.442,76.964,179.9981,-0.0180,-12935.5164
C01209=-93.654,-35.046,76.964,179.9993,-0.0181,-12939.4838
C01210=-95.791,-28.621,76.696,-179.9993,-0.1377,-12943.3646
C01211=-96.473,-22.407,76.288,179.2397,-1.9299,-12946.9242
C01212=-94.154,-17.016,75.883,176.8342,-2.8344,-12949.7558
C01213=-89.334,-13.550,75.383,173.4296,-1.3094,-12951.3752
C01214=-82.740,-12.382,74.428,173.2591,-0.1124,-12951.4889
C01215=-75.576,-11.418,72.474,174.2120,-0.0836,-12951.4087
C01216=-69.129,-10.544,69.894,175.6880,-0.1257,-12951.3277
C01217=-64.262,-9.686,67.375,179.1259,-0.0711,-12951.4285
C01218=-61.417,-8.195,65.554,-162.6105,15.8904,-12952.3998
C01219=-60.695,-4.967,64.832,-173.7605,34.4682,-12955.3216
C01220=-60.785,-2.212,64.801,179.7074,35.5593,-12957.9159
C01221=-60.820,0.000,64.822,-180.0000,35.5497,-12960.0000
C01222=-60.785,2.212,64.801,-179.7074,35.5593,-12962.0841
C01223=-60.695,4.967,64.832,173.7605,34.4682,-12964.6784
C01224=-61.417,8.195,65.554,162.6105,15.8904,-12967.6002
C01225=-64.262,9.686,67.375,-179.1259,-0.0711,-12968.5715
C01226=-69.129,10.544,69.894,-175.6880,-0.1257,-12968.6723
C01227=-75.576,11.418,72.474,-174.2120,-0.0836,-12968.5913
C01228=-82.740,12.382,74.428,-173.2591,-0.1124,-12968.5111
C01229=-89.334,13.550,75.383,-173.4296,-1.3094,-12968.6248
C01230=-94.154,17.016,75.883,-176.8342,-2.8344,-12970.2442
C01231=-96.473,22.407,76.288,-179.2397,-1.9299,-12973.0758
C01232=-95.791,28.621,76.696,179.9993,-0.1377,-12976.6354
C01233=-93.654,35.046,76.964,-179.9993,-0.0181,-12980.5162
C01234=-91.005,41.442,76.964,-179.9981,-0.0180,-12984.4836
C01235=-87.973,47.497,76.696,-179.9983,-0.1358,-12988.3648
C01236=-84.060,52.372,76.288,179.2407,-1.9248,-12991.9242
C01237=-78.609,54.545,75.883,176.8367,-2.8312,-12994.7559
C01238=-72.750,53.588,75.383,173.4272,-1.3089,-12996.3755
C01239=-67.261,49.751,74.428,173.2583,-0.1085,-12996.4893
C01240=-61.514,45.367,72.474,174.2127,-0.0823,-12996.4090
C01241=-56.337,41.426,69.894,175.6860,-0.1257,-12996.3280
C01242=-52.289,38.591,67.375,179.1285,-0.0735,-12996.4285
C01243=-49.223,37.634,65.554,-162.6128,15.8893,-12997.4001
C01244=-46.429,39.406,64.832,-173.7617,34.4707,-13000.3225
C01245=-44.545,41.417,64.801,179.7113,35.5606,-13002.9160
C01246=-43.006,43.006,64.822,-180.0000,35.5489,-13005.0000
C01247=-41.417,44.545,64.801,-179.7113,35.5606,-13007.0840
C01248=-39.405,46.430,64.832,173.7564,34.4670,-13009.6788
C01249=-37.634,49.223,65.554,162.6128,15.8893,-13012.5999
C01250=-38.591,52.289,67.375,-179.1285,-0.0735,-13013.5715
C01251=-41.426,56.337,69.894,-175.6860,-0.1257,-13013.6720
C01252=-45.367,61.514,72.474,-174.2127,-0.0823,-13013.5910
C01253=-49.751,67.261,74.428,-173.2583,-0.1085,-13013.5107
C01254=-53.588,72.750,75.383,-173.4272,-1.3089,-13013.6245
C01255=-54.545,78.609,75.883,-176.8367,-2.8312,-13015.2441
C01256=-52.372,84.060,76.288,-179.2407,-1.9248,-13018.0758
C01257=-47.497,87.973,76.696,179.9983,-0.1358,-13021.6352
C01258=-41.442,91.005,76.964,179.9981,-0.0180,-13025.5164
C01259=-35.046,93.654,76.964,179.9993,-0.0181,-13029.4838
C01260=-28.621,95.791,76.696,-179.9993,-0.1377,-13033.3646
C01261=-22.407,96.473,76.288,179.2397,-1.9299,-13036.9242
C01262=-17.016,94.154,75.883,176.8342,-2.8344,-13039.7558
C01263=-13.550,89.334,75.383,173.4296,-1.3094,-13041.3752
C01264=-12.382,82.740,74.428,173.2591,-0.1124,-13041.4889
C01265=-11.418,75.576,72.474,174.2120,-0.0836,-13041.4087
C01266=-10.544,69.129,69.894,175.6880,-0.1257,-13041.3277
C01267=-9.686,64.262,67.375,179.1259,-0.0711,-13041.4285
C01268=-8.195,61.417,65.554,-162.6105,15.8904,-13042.3998
C01269=-4.967,60.695,64.832,-173.7605,34.4682,-13045.3216
C01270=-2.212,60.785,64.801,179.7074,35.5593,-13047.9159
C01271=0.000,60.820,64.822,-180.0000,35.5497,-13050.0000
C01272=0.000,59.554,66.621,-180.0000,34.6578,-13050.0000
C01273=2.097,59.523,66.599,-179.7230,34.6655,-13052.0177
C01274=4.772,59.445,66.632,173.6798,33.4987,-13054.5896
C01275=7.959,60.221,67.386,163.3494,14.5335,-13057.5288
C01276=9.406,63.206,69.285,-178.7004,-0.0905,-13058.4644
C01277=10.239,68.282,71.901,-175.7112,-0.0994,-13058.5281
C01278=11.109,74.974,74.567,-174.4741,-0.0631,-13058.4283
C01279=12.073,82.372,76.575,-173.6811,-0.0780,-13058.3383
C01280=13.226,89.158,77.551,-173.8761,-1.1797,-13058.4379
C01281=16.717,94.118,78.062,-177.0287,-2.6199,-13060.0717
C01282=22.174,96.515,78.476,-179.2889,-1.7890,-13062.9390
C01283=28.477,95.839,78.891,-179.9987,-0.1251,-13066.5485
C01284=34.998,93.673,79.163,179.9986,-0.0127,-13070.4866
C01285=41.489,90.984,79.163,179.9995,-0.0128,-13074.5131
C01286=47.632,87.904,78.891,179.9965,-0.1257,-13078.4517
C01287=52.567,83.926,78.476,179.2889,-1.7910,-13082.0609
C01288=54.731,78.373,78.062,177.0289,-2.6213,-13084.9281
C01289=53.692,72.396,77.551,173.8708,-1.1760,-13086.5622
C01290=49.709,66.782,76.575,173.6819,-0.0796,-13086.6621
C01291=45.159,60.870,74.567,174.4737,-0.0632,-13086.5714
C01292=41.042,55.523,71.901,175.7117,-0.1034,-13086.4714
C01293=38.042,51.344,69.285,178.6998,-0.0933,-13086.5356
C01294=36.955,48.211,67.386,-163.3536,14.5351,-13087.4711
C01295=38.660,45.408,66.632,-173.6783,33.4962,-13090.4108
C01296=40.607,43.572,66.599,179.7247,34.6655,-13092.9827
C01297=42.111,42.111,66.621,-180.0000,34.6557,-13095.0000
C01298=43.571,40.607,66.599,-179.7195,34.6689,-13097.0166
C01299=45.409,38.659,66.632,173.6775,33.4961,-13099.5906
C01300=48.211,36.955,67.386,163.3501,14.5305,-13102.5289
C01301=51.344,38.042,69.285,-178.6998,-0.0933,-13103.4644
C01302=55.523,41.042,71.901,-175.7117,-0.1034,-13103.5286
C01303=60.870,45.159,74.567,-174.4737,-0.0632,-13103.4286
C01304=66.782,49.709,76.575,-173.6819,-0.0796,-13103.3379
C01305=72.396,53.692,77.551,-173.8708,-1.1760,-13103.4378
C01306=78.373,54.731,78.062,-177.0289,-2.6213,-13105.0719
C01307=83.926,52.567,78.476,-179.2889,-1.7910,-13107.9391
C01308=87.904,47.632,78.891,-179.9965,-0.1257,-13111.5483
C01309=90.984,41.489,79.163,-179.9995,-0.0128,-13115.4869
C01310=93.673,34.998,79.163,-179.9986,-0.0127,-13119.5134
C01311=95.839,28.477,78.891,179.9987,-0.1251,-13123.4515
C01312=96.515,22.174,78.476,179.2889,-1.7890,-13127.0610
C01313=94.118,16.717,78.062,177.0287,-2.6199,-13129.9283
C01314=89.158,13.226,77.551,173.8761,-1.1797,-13131.5621
C01315=82.372,12.073,76.575,173.6811,-0.0780,-13131.6617
C01316=74.974,11.109,74.567,174.4741,-0.0631,-13131.5717
C01317=68.282,10.239,71.901,175.7112,-0.0994,-13131.4719
C01318=63.206,9.406,69.285,178.7004,-0.0905,-13131.5356
C01319=60.221,7.959,67.386,-163.3494,14.5335,-13132.4712
C01320=59.445,4.772,66.632,-173.6798,33.4987,-13135.4104
C01321=59.523,2.097,66.599,179.7230,34.6655,-13137.9823
C01322=59.554,0.000,66.621,180.0000,34.6578,-13140.0000
C01323=59.523,-2.096,66.599,-179.7223,34.6655,-13142.0167
C01324=59.445,-4.772,66.632,173.6803,33.4939,-13144.5896
C01325=60.222,-7.959,67.386,163.3494,14.5335,-13147.5286
C01326=63.206,-9.406,69.285,-178.7004,-0.0905,-13148.4644
C01327=68.282,-10.239,71.901,-175.7112,-0.0994,-13148.5281
C01328=74.974,-11.109,74.567,-174.4741,-0.0631,-13148.4283
C01329=82.372,-12.073,76.575,-173.6811,-0.0780,-13148.3383
C01330=89.158,-13.226,77.551,-173.8761,-1.1797,-13148.4379
C01331=94.118,-16.717,78.062,-177.0287,-2.6199,-13150.0717
C01332=96.515,-22.174,78.476,-179.2889,-1.7890,-13152.9390
C01333=95.839,-28.477,78.891,-179.9987,-0.1251,-13156.5485
C01334=93.673,-34.998,79.163,179.9986,-0.0127,-13160.4866
C01335=90.984,-41.489,79.163,179.9995,-0.0128,-13164.5131
C01336=87.904,-47.632,78.891,179.9965,-0.1257,-13168.4517
C01337=83.926,-52.567,78.476,179.2889,-1.7910,-13172.0609
C01338=78.373,-54.731,78.062,177.0289,-2.6213,-13174.9281
C01339=72.396,-53.692,77.551,173.8708,-1.1760,-13176.5622
C01340=66.782,-49.709,76.575,173.6819,-0.0796,-13176.6621
C01341=60.870,-45.159,74.567,174.4737,-0.0632,-13176.5714
C01342=55.523,-41.042,71.901,175.7117,-0.1034,-13176.4714
C01343=51.344,-38.042,69.285,178.6998,-0.0933,-13176.5356
C01344=48.211,-36.955,67.386,-163.3536,14.5351,-13177.4711
C01345=45.408,-38.660,66.632,-173.6783,33.4962,-13180.4108
C01346=43.572,-40.607,66.599,179.7247,34.6655,-13182.9827
C01347=42.111,-42.111,66.621,180.0000,34.6557,-13185.0000
C01348=40.607,-43.571,66.599,-179.7195,34.6689,-13187.0166
C01349=38.659,-45.409,66.632,173.6775,33.4961,-13189.5906
C01350=36.955,-48.211,67.386,163.3501,14.5305,-13192.5289
C01351=38.042,-51.344,69.285,-178.6998,-0.0933,-13193.4644
C01352=41.042,-55.523,71.901,-175.7117,-0.1034,-13193.5286
C01353=45.159,-60.870,74.567,-174.4737,-0.0632,-13193.4286
C01354=49.709,-66.782,76.575,-173.6819,-0.0796,-13193.3379
C01355=53.692,-72.396,77.551,-173.8708,-1.1760,-13193.4378
C01356=54.731,-78.373,78.062,-177.0289,-2.6213,-13195.0719
C01357=52.567,-83.926,78.476,-179.2889,-1.7910,-13197.9391
C01358=47.632,-87.904,78.891,-179.9965,-0.1257,-13201.5483
C01359=41.489,-90.984,79.163,-179.9995,-0.0128,-13205.4869
C01360=34.998,-93.673,79.163,-179.9986,-0.0127,-13209.5134
C01361=28.477,-95.839,78.891,179.9987,-0.1251,-13213.4515
C01362=22.174,-96.515,78.476,179.2889,-1.7890,-13217.0610
C01363=16.717,-94.118,78.062,177.0287,-2.6199,-13219.9283
C01364=13.226,-89.158,77.551,173.8761,-1.1797,-13221.5621
C01365=12.073,-82.372,76.575,173.6811,-0.0780,-13221.6617
C01366=11.109,-74.974,74.567,174.4741,-0.0631,-13221.5717
C01367=10.239,-68.282,71.901,175.7112,-0.0994,-13221.4719
C01368=9.406,-63.206,69.285,178.7004,-0.0905,-13221.5356
C01369=7.959,-60.221,67.386,-163.3494,14.5335,-13222.4712
C01370=4.772,-59.445,66.632,-173.6798,33.4987,-13225.4104
C01371=2.097,-59.523,66.599,179.7230,34.6655,-13227.9823
C01372=0.000,-59.554,66.621,180.0000,34.6578,-13230.0000
C01373=0.000,-59.554,66.621,180.0000,34.6578,-13230.0000
C01374=-2.096,-59.523,66.599,-179.7223,34.6655,-13232.0167
C01375=-4.772,-59.445,66.632,173.6803,33.4939,-13234.5896
C01376=-7.959,-60.222,67.386,163.3494,14.5335,-13237.5286
C01377=-9.406,-63.206,69.285,-178.7004,-0.0905,-13238.4644
C01378=-10.239,-68.282,71.901,-175.7112,-0.0994,-13238.5281
C01379=-11.109,-74.974,74.567,-174.4741,-0.0631,-13238.4283
C01380=-12.073,-82.372,76.575,-173.6811,-0.0780,-13238.3383
C01381=-13.226,-89.158,77.551,-173.8761,-1.1797,-13238.4379
C01382=-16.717,-94.118,78.062,-177.0287,-2.6199,-13240.0717
C01383=-22.174,-96.515,78.476,-179.2889,-1.7890,-13242.9390
C01384=-28.477,-95.839,78.891,-179.9987,-0.1251,-13246.5485
C01385=-34.998,-93.673,79.163,179.9986,-0.0127,-13250.4866
C01386=-41.489,-90.984,79.163,179.9995,-0.0128,-13254.5131
C01387=-47.632,-87.904,78.891,179.9965,-0.1257,-13258.4517
C01388=-52.567,-83.926,78.476,179.2889,-1.7910,-13262.0609
C01389=-54.731,-78.373,78.062,177.0289,-2.6213,-13264.9281
C01390=-53.692,-72.396,77.551,173.8708,-1.1760,-13266.5622
C01391=-49.709,-66.782,76.575,173.6819,-0.0796,-13266.6621
C01392=-45.159,-60.870,74.567,174.4737,-0.0632,-13266.5714
C01393=-41.042,-55.523,71.901,175.7117,-0.1034,-13266.4714
C01394=-38.042,-51.344,69.285,178.6998,-0.0933,-13266.5356
C01395=-36.955,-48.211,67.386,-163.3536,14.5351,-13267.4711
C01396=-38.660,-45.408,66.632,-173.6783,33.4962,-13270.4108
C01397=-40.607,-43.572,66.599,179.7247,34.6655,-13272.9827
C01398=-42.111,-42.111,66.621,180.0000,34.6557,-13275.0000
C01399=-43.571,-40.607,66.599,-179.7195,34.6689,-13277.0166
C01400=-45.409,-38.659,66.632,173.6775,33.4961,-13279.5906
C01401=-48.211,-36.955,67.386,163.3501,14.5305,-13282.5289
C01402=-51.344,-38.042,69.285,-178.6998,-0.0933,-13283.4644
C01403=-55.523,-41.042,71.901,-175.7117,-0.1034,-13283.5286
C01404=-60.870,-45.159,74.567,-174.4737,-0.0632,-13283.4286
C01405=-66.782,-49.709,76.575,-173.6819,-0.0796,-13283.3379
C01406=-72.396,-53.692,77.551,-173.8708,-1.1760,-13283.4378
C01407=-78.373,-54.731,78.062,-177.0289,-2.6213,-13285.0719
C01408=-83.926,-52.567,78.476,-179.2889,-1.7910,-13287.9391
C01409=-87.904,-47.632,78.891,-179.9965,-0.1257,-13291.5483
C01410=-90.984,-41.489,79.163,-179.9995,-0.0128,-13295.4869
C01411=-93.673,-34.998,79.163,-179.9986,-0.0127,-13299.5134
C01412=-95.839,-28.477,78.891,179.9987,-0.1251,-13303.4515
C01413=-96.515,-22.174,78.476,179.2889,-1.7890,-13307.0610
C01414=-94.118,-16.717,78.062,177.0287,-2.6199,-13309.9283
C01415=-89.158,-13.226,77.551,173.8761,-1.1797,-13311.5621
C01416=-82.372,-12.073,76.575,173.6811,-0.0780,-13311.6617
C01417=-74.974,-11.109,74.567,174.4741,-0.0631,-13311.5717
C01418=-68.282,-10.239,71.901,175.7112,-0.0994,-13311.4719
C01419=-63.206,-9.406,69.285,178.7004,-0.0905,-13311.5356
C01420=-60.221,-7.959,67.386,-163.3494,14.5335,-13312.4712
C01421=-59.445,-4.772,66.632,-173.6798,33.4987,-13315.4104
C01422=-59.523,-2.097,66.599,179.7230,34.6655,-13317.9823
C01423=-59.554,0.000,66.621,-180.0000,34.6578,-13320.0000
C01424=-59.523,2.096,66.599,-179.7223,34.6655,-13322.0167
C01425=-59.445,4.772,66.632,173.6803,33.4939,-13324.5896
C01426=-60.222,7.959,67.386,163.3494,14.5335,-13327.5286
C01427=-63.206,9.406,69.285,-178.7004,-0.0905,-13328.4644
C01428=-68.282,10.239,71.901,-175.7112,-0.0994,-13328.5281
C01429=-74.974,11.109,74.567,-174.4741,-0.0631,-13328.4283
C01430=-82.372,12.073,76.575,-173.6811,-0.0780,-13328.3383
C01431=-89.158,13.226,77.551,-173.8761,-1.1797,-13328.4379
C01432=-94.118,16.717,78.062,-177.0287,-2.6199,-13330.0717
C01433=-96.515,22.174,78.476,-179.2889,-1.7890,-13332.9390
C01434=-95.839,28.477,78.891,-179.9987,-0.1251,-13336.5485
C01435=-93.673,34.998,79.163,179.9986,-0.0127,-13340.4866
C01436=-90.984,41.489,79.163,179.9995,-0.0128,-13344.5131
C01437=-87.904,47.632,78.891,179.9965,-0.1257,-13348.4517
C01438=-83.926,52.567,78.476,179.2889,-1.7910,-13352.0609
C01439=-78.373,54.731,78.062,177.0289,-2.6213,-13354.9281
C01440=-72.396,53.692,77.551,173.8708,-1.1760,-13356.5622
C01441=-66.782,49.709,76.575,173.6819,-0.0796,-13356.6621
C01442=-60.870,45.159,74.567,174.4737,-0.0632,-13356.5714
C01443=-55.523,41.042,71.901,175.7117,-0.1034,-13356.4714
C01444=-51.344,38.042,69.285,178.6998,-0.0933,-13356.5356
C01445=-48.211,36.955,67.386,-163.3536,14.5351,-13357.4711
C01446=-45.408,38.660,66.632,-173.6783,33.4962,-13360.4108
C01447=-43.572,40.607,66.599,179.7247,34.6655,-13362.9827
C01448=-42.111,42.111,66.621,-180.0000,34.6557,-13365.0000
C01449=-40.607,43.571,66.599,-179.7195,34.6689,-13367.0166
C01450=-38.659,45.409,66.632,173.6775,33.4961,-13369.5906
C01451=-36.955,48.211,67.386,163.3501,14.5305,-13372.5289
C01452=-38.042,51.344,69.285,-178.6998,-0.0933,-13373.4644
C01453=-41.042,55.523,71.901,-175.7117,-0.1034,-13373.5286
C01454=-45.159,60.870,74.567,-174.4737,-0.0632,-13373.4286
C01455=-49.709,66.782,76.575,-173.6819,-0.0796,-13373.3379
C01456=-53.692,72.396,77.551,-173.8708,-1.1760,-13373.4378
C01457=-54.731,78.373,78.062,-177.0289,-2.6213,-13375.0719
C01458=-52.567,83.926,78.476,-179.2889,-1.7910,-13377.9391
C01459=-47.632,87.904,78.891,-179.9965,-0.1257,-13381.5483
C01460=-41.489,90.984,79.163,-179.9995,-0.0128,-13385.4869
C01461=-34.998,93.673,79.163,-179.9986,-0.0127,-13389.5134
C01462=-28.477,95.839,78.891,179.9987,-0.1251,-13393.4515
C01463=-22.174,96.515,78.476,179.2889,-1.7890,-13397.0610
C01464=-16.717,94.118,78.062,177.0287,-2.6199,-13399.9283
C01465=-13.226,89.158,77.551,173.8761,-1.1797,-13401.5621
C01466=-12.073,82.372,76.575,173.6811,-0.0780,-13401.6617
C01467=-11.109,74.974,74.567,174.4741,-0.0631,-13401.5717
C01468=-10.239,68.282,71.901,175.7112,-0.0994,-13401.4719
C01469=-9.406,63.206,69.285,178.7004,-0.0905,-13401.5356
C01470=-7.959,60.222,67.386,-163.3494,14.5335,-13402.4714
C01471=-4.772,59.445,66.632,-173.6803,33.4939,-13405.4104
C01472=-2.096,59.523,66.599,179.7223,34.6655,-13407.9833
C01473=0.000,59.554,66.621,-180.0000,34.6578,-13410.0000
C01474=0.000,58.319,68.442,-180.0000,33.6424,-13410.0000
C01475=1.984,58.291,68.419,-179.7349,33.6528,-13411.9494
C01476=4.582,58.225,68.453,173.6435,32.4018,-13414.4996
C01477=7.730,59.058,69.238,164.1787,13.2130,-13417.4570
C01478=9.135,62.185,71.215,-178.3577,-0.1005,-13418.3570
C01479=9.949,67.473,73.927,-175.8025,-0.0826,-13418.3879
C01480=10.820,74.409,76.674,-174.7933,-0.0431,-13418.2735
C01481=11.787,82.032,78.729,-174.1646,-0.0547,-13418.1767
C01482=12.929,88.996,79.725,-174.3851,-1.0436,-13418.2659
C01483=16.445,94.085,80.245,-177.2659,-2.3820,-13419.9145
C01484=21.964,96.553,80.665,-179.3477,-1.6266,-13422.8156
C01485=28.347,95.882,81.086,179.9979,-0.1141,-13426.4700
C01486=34.955,93.690,81.363,179.9986,-0.0127,-13430.4601
C01487=41.532,90.965,81.363,179.9995,-0.0128,-13434.5401
C01488=47.755,87.843,81.086,179.9989,-0.1180,-13438.5303
C01489=52.743,83.804,80.665,179.3513,-1.6270,-13442.1847
C01490=54.900,78.157,80.245,177.2696,-2.3811,-13445.0854
C01491=53.787,72.072,79.725,174.3816,-1.0449,-13446.7338
C01492=49.670,66.340,78.729,174.1696,-0.0563,-13446.8229
C01493=44.964,60.266,76.674,174.7950,-0.0468,-13446.7263
C01494=40.676,54.746,73.927,175.8029,-0.0822,-13446.6122
C01495=37.512,50.430,71.215,178.3596,-0.0990,-13446.6435
C01496=36.294,47.226,69.238,-164.1774,13.2171,-13447.5429
C01497=37.931,44.411,68.453,-173.6447,32.4038,-13450.5003
C01498=39.816,42.621,68.419,179.7347,33.6545,-13453.0512
C01499=41.238,41.238,68.442,-180.0000,33.6466,-13455.0000
C01500=42.621,39.816,68.419,-179.7347,33.6545,-13456.9488
C01501=44.412,37.931,68.453,173.6400,32.4000,-13459.5003
C01502=47.226,36.294,69.238,164.1774,13.2171,-13462.4571
C01503=50.430,37.512,71.215,-178.3596,-0.0990,-13463.3565
C01504=54.746,40.676,73.927,-175.8029,-0.0822,-13463.3878
C01505=60.266,44.964,76.674,-174.7950,-0.0468,-13463.2737
C01506=66.340,49.670,78.729,-174.1696,-0.0563,-13463.1771
C01507=72.072,53.787,79.725,-174.3816,-1.0449,-13463.2662
C01508=78.157,54.900,80.245,-177.2696,-2.3811,-13464.9146
C01509=83.804,52.743,80.665,-179.3513,-1.6270,-13467.8153
C01510=87.843,47.755,81.086,-179.9989,-0.1180,-13471.4697
C01511=90.965,41.532,81.363,-179.9995,-0.0128,-13475.4599
C01512=93.690,34.955,81.363,-179.9986,-0.0127,-13479.5399
C01513=95.882,28.347,81.086,-179.9979,-0.1141,-13483.5300
C01514=96.553,21.964,80.665,179.3477,-1.6266,-13487.1844
C01515=94.085,16.445,80.245,177.2659,-2.3820,-13490.0855
C01516=88.996,12.929,79.725,174.3851,-1.0436,-13491.7341
C01517=82.032,11.787,78.729,174.1646,-0.0547,-13491.8233
C01518=74.409,10.820,76.674,174.7933,-0.0431,-13491.7265
C01519=67.473,9.949,73.927,175.8025,-0.0826,-13491.6121
C01520=62.185,9.135,71.215,178.3577,-0.1005,-13491.6430
C01521=59.058,7.730,69.238,-164.1787,13.2130,-13492.5430
C01522=58.225,4.582,68.453,-173.6435,32.4018,-13495.5004
C01523=58.291,1.984,68.419,179.7349,33.6528,-13498.0506
C01524=58.319,0.000,68.442,-180.0000,33.6424,-13500.0000
C01525=58.291,-1.983,68.419,-179.7342,33.6528,-13501.9484
C01526=58.225,-4.583,68.453,173.6429,32.4017,-13504.5006
C01527=59.058,-7.730,69.238,164.1787,13.2130,-13507.4570
C01528=62.185,-9.135,71.215,-178.3577,-0.1005,-13508.3570
C01529=67.473,-9.949,73.927,-175.8025,-0.0826,-13508.3879
C01530=74.409,-10.820,76.674,-174.7933,-0.0431,-13508.2735
C01531=82.032,-11.787,78.729,-174.1646,-0.0547,-13508.1767
C01532=88.996,-12.929,79.725,-174.3851,-1.0436,-13508.2659
C01533=94.085,-16.445,80.245,-177.2659,-2.3820,-13509.9145
C01534=96.553,-21.964,80.665,-179.3477,-1.6266,-13512.8156
C01535=95.882,-28.347,81.086,179.9979,-0.1141,-13516.4700
C01536=93.690,-34.955,81.363,179.9986,-0.0127,-13520.4601
C01537=90.965,-41.532,81.363,179.9995,-0.0128,-13524.5401
C01538=87.843,-47.755,81.086,179.9989,-0.1180,-13528.5303
C01539=83.804,-52.743,80.665,179.3513,-1.6270,-13532.1847
C01540=78.157,-54.900,80.245,177.2696,-2.3811,-13535.0854
C01541=72.072,-53.787,79.725,174.3816,-1.0449,-13536.7338
C01542=66.340,-49.670,78.729,174.1696,-0.0563,-13536.8229
C01543=60.266,-44.964,76.674,174.7950,-0.0468,-13536.7263
C01544=54.746,-40.676,73.927,175.8029,-0.0822,-13536.6122
C01545=50.430,-37.512,71.215,178.3596,-0.0990,-13536.6435
C01546=47.226,-36.294,69.238,-164.1774,13.2171,-13537.5429
C01547=44.411,-37.931,68.453,-173.6447,32.4038,-13540.5003
C01548=42.621,-39.816,68.419,179.7347,33.6545,-13543.0512
C01549=41.238,-41.238,68.442,-180.0000,33.6466,-13545.0000
C01550=39.816,-42.621,68.419,-179.7347,33.6545,-13546.9488
C01551=37.931,-44.412,68.453,173.6400,32.4000,-13549.5003
C01552=36.294,-47.226,69.238,164.1774,13.2171,-13552.4571
C01553=37.512,-50.430,71.215,-178.3596,-0.0990,-13553.3565
C01554=40.676,-54.746,73.927,-175.8029,-0.0822,-13553.3878
C01555=44.964,-60.266,76.674,-174.7950,-0.0468,-13553.2737
C01556=49.670,-66.340,78.729,-174.1696,-0.0563,-13553.1771
C01557=53.787,-72.072,79.725,-174.3816,-1.0449,-13553.2662
C01558=54.900,-78.157,80.245,-177.2696,-2.3811,-13554.9146
C01559=52.743,-83.804,80.665,-179.3513,-1.6270,-13557.8153
C01560=47.755,-87.843,81.086,-179.9989,-0.1180,-13561.4697
C01561=41.532,-90.965,81.363,-179.9995,-0.0128,-13565.4599
C01562=34.955,-93.690,81.363,-179.9986,-0.0127,-13569.5399
C01563=28.347,-95.882,81.086,-179.9979,-0.1141,-13573.5300
C01564=21.964,-96.553,80.665,179.3477,-1.6266,-13577.1844
C01565=16.445,-94.085,80.245,177.2659,-2.3820,-13580.0855
C01566=12.929,-88.996,79.725,174.3851,-1.0436,-13581.7341
C01567=11.787,-82.032,78.729,174.1646,-0.0547,-13581.8233
C01568=10.820,-74.409,76.674,174.7933,-0.0431,-13581.7265
C01569=9.949,-67.473,73.927,175.8025,-0.0826,-13581.6121
C01570=9.135,-62.185,71.215,178.3577,-0.1005,-13581.6430
C01571=7.730,-59.058,69.238,-164.1787,13.2130,-13582.5430
C01572=4.582,-58.225,68.453,-173.6435,32.4018,-13585.5004
C01573=1.984,-58.291,68.419,179.7349,33.6528,-13588.0506
C01574=0.000,-58.319,68.442,-180.0000,33.6424,-13590.0000
C01575=0.000,-58.319,68.442,-180.0000,33.6424,-13590.0000
C01576=-1.983,-58.291,68.419,-179.7342,33.6528,-13591.9484
C01577=-4.583,-58.225,68.453,173.6429,32.4017,-13594.5006
C01578=-7.730,-59.058,69.238,164.1787,13.2130,-13597.4570
C01579=-9.135,-62.185,71.215,-178.3577,-0.1005,-13598.3570
C01580=-9.949,-67.473,73.927,-175.8025,-0.0826,-13598.3879
C01581=-10.820,-74.409,76.674,-174.7933,-0.0431,-13598.2735
C01582=-11.787,-82.032,78.729,-174.1646,-0.0547,-13598.1767
C01583=-12.929,-88.996,79.725,-174.3851,-1.0436,-13598.2659
C01584=-16.445,-94.085,80.245,-177.2659,-2.3820,-13599.9145
C01585=-21.964,-96.553,80.665,-179.3477,-1.6266,-13602.8156
C01586=-28.347,-95.882,81.086,179.9979,-0.1141,-13606.4700
C01587=-34.955,-93.690,81.363,179.9986,-0.0127,-13610.4601
C01588=-41.532,-90.965,81.363,179.9995,-0.0128,-13614.5401
C01589=-47.755,-87.843,81.086,179.9989,-0.1180,-13618.5303
C01590=-52.743,-83.804,80.665,179.3513,-1.6270,-13622.1847
C01591=-54.900,-78.157,80.245,177.2696,-2.3811,-13625.0854
C01592=-53.787,-72.072,79.725,174.3816,-1.0449,-13626.7338
C01593=-49.670,-66.340,78.729,174.1696,-0.0563,-13626.8229
C01594=-44.964,-60.266,76.674,174.7950,-0.0468,-13626.7263
C01595=-40.676,-54.746,73.927,175.8029,-0.0822,-13626.6122
C01596=-37.512,-50.430,71.215,178.3596,-0.0990,-13626.6435
C01597=-36.294,-47.226,69.238,-164.1774,13.2171,-13627.5429
C01598=-37.931,-44.411,68.453,-173.6447,32.4038,-13630.5003
C01599=-39.816,-42.621,68.419,179.7347,33.6545,-13633.0512
C01600=-41.238,-41.238,68.442,180.0000,33.6466,-13635.0000
C01601=-42.621,-39.816,68.419,-179.7347,33.6545,-13636.9488
C01602=-44.412,-37.931,68.453,173.6400,32.4000,-13639.5003
C01603=-47.226,-36.294,69.238,164.1774,13.2171,-13642.4571
C01604=-50.430,-37.512,71.215,-178.3596,-0.0990,-13643.3565
C01605=-54.746,-40.676,73.927,-175.8029,-0.0822,-13643.3878
C01606=-60.266,-44.964,76.674,-174.7950,-0.0468,-13643.2737
C01607=-66.340,-49.670,78.729,-174.1696,-0.0563,-13643.1771
C01608=-72.072,-53.787,79.725,-174.3816,-1.0449,-13643.2662
C01609=-78.157,-54.900,80.245,-177.2696,-2.3811,-13644.9146
C01610=-83.804,-52.743,80.665,-179.3513,-1.6270,-13647.8153
C01611=-87.843,-47.755,81.086,-179.9989,-0.1180,-13651.4697
C01612=-90.965,-41.532,81.363,-179.9995,-0.0128,-13655.4599
C01613=-93.690,-34.955,81.363,-179.9986,-0.0127,-13659.5399
C01614=-95.882,-28.347,81.086,-179.9979,-0.1141,-13663.5300
C01615=-96.553,-21.964,80.665,179.3477,-1.6266,-13667.1844
C01616=-94.085,-16.445,80.245,177.2659,-2.3820,-13670.0855
C01617=-88.996,-12.929,79.725,174.3851,-1.0436,-13671.7341
C01618=-82.032,-11.787,78.729,174.1646,-0.0547,-13671.8233
C01619=-74.409,-10.820,76.674,174.7933,-0.0431,-13671.7265
C01620=-67.473,-9.949,73.927,175.8025,-0.0826,-13671.6121
C01621=-62.185,-9.135,71.215,178.3577,-0.1005,-13671.6430
C01622=-59.058,-7.730,69.238,-164.1787,13.2130,-13672.5430
C01623=-58.225,-4.582,68.453,-173.6435,32.4018,-13675.5004
C01624=-58.291,-1.984,68.419,179.7349,33.6528,-13678.0506
C01625=-58.319,0.000,68.442,180.0000,33.6424,-13680.0000
C01626=-58.291,1.983,68.419,-179.7342,33.6528,-13681.9484
C01627=-58.225,4.583,68.453,173.6429,32.4017,-13684.5006
C01628=-59.058,7.730,69.238,164.1787,13.2130,-13687.4570
C01629=-62.185,9.135,71.215,-178.3577,-0.1005,-13688.3570
C01630=-67.473,9.949,73.927,-175.8025,-0.0826,-13688.3879
C01631=-74.409,10.820,76.674,-174.7933,-0.0431,-13688.2735
C01632=-82.032,11.787,78.729,-174.1646,-0.0547,-13688.1767
C01633=-88.996,12.929,79.725,-174.3851,-1.0436,-13688.2659
C01634=-94.085,16.445,80.245,-177.2659,-2.3820,-13689.9145
C01635=-96.553,21.964,80.665,-179.3477,-1.6266,-13692.8156
C01636=-95.882,28.347,81.086,179.9979,-0.1141,-13696.4700
C01637=-93.690,34.955,81.363,179.9986,-0.0127,-13700.4601
C01638=-90.965,41.532,81.363,179.9995,-0.0128,-13704.5401
C01639=-87.843,47.755,81.086,179.9989,-0.1180,-13708.5303
C01640=-83.804,52.743,80.665,179.3513,-1.6270,-13712.1847
C01641=-78.157,54.900,80.245,177.2696,-2.3811,-13715.0854
C01642=-72.072,53.787,79.725,174.3816,-1.0449,-13716.7338
C01643=-66.340,49.670,78.729,174.1696,-0.0563,-13716.8229
C01644=-60.266,44.964,76.674,174.7950,-0.0468,-13716.7263
C01645=-54.746,40.676,73.927,175.8029,-0.0822,-13716.6122
C01646=-50.430,37.512,71.215,178.3596,-0.0990,-13716.6435
C01647=-47.226,36.294,69.238,-164.1774,13.2171,-13717.5429
C01648=-44.411,37.931,68.453,-173.6447,32.4038,-13720.5003
C01649=-42.621,39.816,68.419,179.7347,33.6545,-13723.0512
C01650=-41.238,41.238,68.442,180.0000,33.6466,-13725.0000
C01651=-39.816,42.621,68.419,-179.7347,33.6545,-13726.9488
C01652=-37.931,44.412,68.453,173.6400,32.4000,-13729.5003
C01653=-36.294,47.226,69.238,164.1774,13.2171,-13732.4571
C01654=-37.512,50.430,71.215,-178.3596,-0.0990,-13733.3565
C01655=-40.676,54.746,73.927,-175.8029,-0.0822,-13733.3878
C01656=-44.964,60.266,76.674,-174.7950,-0.0468,-13733.2737
C01657=-49.670,66.340,78.729,-174.1696,-0.0563,-13733.1771
C01658=-53.787,72.072,79.725,-174.3816,-1.0449,-13733.2662
C01659=-54.900,78.157,80.245,-177.2696,-2.3811,-13734.9146
C01660=-52.743,83.804,80.665,-179.3513,-1.6270,-13737.8153
C01661=-47.755,87.843,81.086,-179.9989,-0.1180,-13741.4697
C01662=-41.532,90.965,81.363,-179.9995,-0.0128,-13745.4599
C01663=-34.955,93.690,81.363,-179.9986,-0.0127,-13749.5399
C01664=-28.347,95.882,81.086,-179.9979,-0.1141,-13753.5300
C01665=-21.964,96.553,80.665,179.3477,-1.6266,-13757.1844
C01666=-16.445,94.085,80.245,177.2659,-2.3820,-13760.0855
C01667=-12.929,88.996,79.725,174.3851,-1.0436,-13761.7341
C01668=-11.787,82.032,78.729,174.1646,-0.0547,-13761.8233
C01669=-10.820,74.409,76.674,174.7933,-0.0431,-13761.7265
C01670=-9.949,67.473,73.927,175.8025,-0.0826,-13761.6121
C01671=-9.135,62.185,71.215,178.3577,-0.1005,-13761.6430
C01672=-7.730,59.058,69.238,-164.1787,13.2130,-13762.5430
C01673=-4.583,58.225,68.453,-173.6429,32.4017,-13765.4994
C01674=-1.983,58.291,68.419,179.7342,33.6528,-13768.0516
C01675=0.000,58.319,68.442,-180.0000,33.6424,-13770.0000
C01676=0.000,57.118,70.285,-180.0000,32.4949,-13770.0000
C01677=1.874,57.094,70.261,-179.7573,32.5080,-13771.8799
C01678=4.398,57.039,70.297,173.6555,31.1772,-13774.4091
C01679=7.507,57.930,71.114,165.0758,11.9424,-13777.3837
C01680=8.875,61.204,73.167,-178.1043,-0.0957,-13778.2508
C01681=9.674,66.709,75.971,-175.9523,-0.0621,-13778.2514
C01682=10.553,73.885,78.794,-175.1749,-0.0294,-13778.1286
C01683=11.527,81.722,80.892,-174.7101,-0.0362,-13778.0287
C01684=12.662,88.851,81.904,-174.9556,-0.9120,-13778.1105
C01685=16.202,94.056,82.431,-177.5455,-2.1207,-13779.7738
C01686=21.776,96.587,82.857,-179.4149,-1.4483,-13782.7052
C01687=28.231,95.920,83.283,-180.0000,-0.1015,-13786.4001
C01688=34.916,93.705,83.562,179.9986,-0.0127,-13790.4362
C01689=41.570,90.949,83.562,179.9996,-0.0128,-13794.5637
C01690=47.863,87.788,83.283,179.9986,-0.1052,-13798.5997
C01691=52.900,83.695,82.857,179.4162,-1.4469,-13802.2952
C01692=55.051,77.964,82.431,177.5443,-2.1205,-13805.2262
C01693=53.873,71.781,81.904,174.9523,-0.9140,-13806.8889
C01694=49.635,65.937,80.892,174.7131,-0.0370,-13806.9711
C01695=44.783,59.707,78.794,175.1691,-0.0312,-13806.8716
C01696=40.330,54.011,75.971,175.9514,-0.0603,-13806.7487
C01697=37.003,49.553,73.167,178.1031,-0.0935,-13806.7500
C01698=35.654,46.271,71.114,-165.0753,11.9430,-13807.6160
C01699=37.223,43.442,70.297,-173.6602,31.1794,-13810.5914
C01700=39.047,41.697,70.261,179.7562,32.5069,-13813.1202
C01701=40.388,40.388,70.285,-180.0000,32.4978,-13815.0000
C01702=41.696,39.047,70.261,-179.7558,32.5069,-13816.8791
C01703=43.443,37.223,70.297,173.6555,31.1756,-13819.4092
C01704=46.271,35.654,71.114,165.0753,11.9430,-13822.3840
C01705=49.553,37.003,73.167,-178.1031,-0.0935,-13823.2500
C01706=54.011,40.330,75.971,-175.9514,-0.0603,-13823.2513
C01707=59.707,44.783,78.794,-175.1691,-0.0312,-13823.1284
C01708=65.937,49.635,80.892,-174.7131,-0.0370,-13823.0289
